METHOD PUBLIC finish : BOOL//Return value = TRUE if state was <> 0 and Err.flag = FALSE
VAR_INPUT
END_VAR
IF state <> 0 
THEN
	Busy 													:= FALSE;
	Done 													:= NOT Err.flag;
	     													  													
	text 													:= CONCAT('FINISH~State:',DINT_TO_STRING(state));
	text 													:= CONCAT(text,'(SetState:');
	text 													:= CONCAT(text,DINT_TO_STRING(MemSetState));
	text 													:= CONCAT(text,')/Busy=');
	text 													:= CONCAT(text,BOOL_TO_STRING(Busy));
	text 													:= CONCAT(text,'/Done=');
	text 													:= CONCAT(text,BOOL_TO_STRING(Done));
	
	state													:= 0;
	Finish 													:= Done;	
ELSE
	Finish 													:= FALSE;
END_IF
END_METHOD

METHOD PUBLIC incState : BOOL //Increment State by NoOfIncrements / Result always true 
VAR_INPUT
	NoOfIncrements								:	DINT;
END_VAR
State := State + NoOfIncrements;
incState := TRUE;
END_METHOD

METHOD PUBLIC reset : BOOL //return value = TRUE if execution finished 
VAR_INPUT
END_VAR
Done 														:= FALSE;
Busy 														:= FALSE;
text 														:= CONCAT('RESET~State:',DINT_TO_STRING(state));
text 														:= CONCAT(text,'(SetState:');
text 														:= CONCAT(text,DINT_TO_STRING(MemSetState));
text 														:= CONCAT(text,')/Busy=');
text 														:= CONCAT(text,BOOL_TO_STRING(Busy));
text 														:= CONCAT(text,'/Done=');
text 														:= CONCAT(text,BOOL_TO_STRING(Done));

MemSetState := state 										:=  0;
reset 														:= TRUE;
END_METHOD

METHOD PUBLIC resetWithErrHdl : BOOL //return value = TRUE if execution finished 
VAR_INPUT
END_VAR
Reset();
Err.Reset();
ResetWithErrHdl												 := TRUE;
END_METHOD

METHOD PUBLIC set : BOOL //Set MemSetstate to state value, Return value = TRUE if sequence handle will be busy (State <> 0)
VAR_INPUT
	State													:		 DINT;
END_VAR
MemSetState 												:= THIS^.state := State;
Busy 														:= state <> 0;
Done 														:= FALSE;
Set															:= Busy;
                    										
text 														:= CONCAT('SET~State:',DINT_TO_STRING(MemSetstate));
END_METHOD

PROPERTY PUBLIC ton_BT : TIME
GET
IF ton.IN
	AND NOT ton.Q
THEN
	Ton_BT 													:= ton.PT - ton.ET;
ELSE       													
	Ton_BT 													:= T#0MS;
END_IF
END_GET
END_PROPERTY

PROPERTY PUBLIC ton_PT : TIME
GET
Ton_PT 														:= ton.PT;
END_GET
SET
PUBLIC 
VAR
END_VAR
Ton.PT 														:= Ton_PT;
END_SET
END_PROPERTY

METHOD PUBLIC tonOFF : BOOL //Return value = TRUE if execution finished
VAR_INPUT
END_VAR
TON(In := FALSE,Q => );
TonOFF := NOT Ton.Q;
END_METHOD

METHOD PUBLIC tonON : BOOL; //Return value = TRUE if execution finished
VAR_INPUT
END_VAR
TON(In := TRUE,Q => TonON);
END_METHOD

METHOD PUBLIC tonRUN : BOOL //Return value status of time (Ton.Q)
VAR_INPUT
	IN														:	BOOL;
	PT														:	TIME;
END_VAR
THIS^.TON.IN := IN;
THIS^.TON.PT := PT;
TON(IN := IN , PT := PT, Q => TonRUN);
END_METHOD

END_FUNCTION_BLOCK

// POUs/_Miscellaneous/setNoOfBits
//Returns a LWORD variable with number (no) of bits set to TRUE starting from lowest significant bit (.0)  
{attribute 'displaymode':='binary'}		
FUNCTION setNoOfBits : LWORD 
VAR_INPUT
	No														:	INT;
END_VAR
VAR
	u64														:	U_64BIT_DATATYPE;
END_VAR

IF No <= 0
THEN
	setNoOfBits												:= 0;
ELSIF No <= 32
THEN
	setNoOfBits												:= TO_LWORD((EXPT(2,No) - 1));
ELSE
	u64._DWORDs[0]											:= 16#FFFFFFFF;
	u64._DWORDs[1]											:= TO_DWORD((EXPT(2,No - 32) - 1));
	setNoOfBits												:= u64._LWORD;
END_IF

END_FUNCTION

// POUs/_Miscellaneous/TEST_FB
//Should be called after new FBs to test signal flow and behavior of PlcOpen related variables 
FUNCTION_BLOCK Test_FB
VAR_OUTPUT CONSTANT
	NO_ERR 													:	INT := 0;
 	OK														:	INT := 1;
	ERR_BUSY 												:	INT := 2;
	ERR_DONE 												:	INT := 3;	
	ERR_ERR 												:	INT := 4;
	ERR_DONE_ERROR											:	INT := 5;
	ERR_NO_SIGNAL											:	INT := 6;
END_VAR             										
VAR_INPUT           										
	Reset													:	BOOL;	//The function block will be reset with a rising edge 
	Execute													:	BOOL;	//Link with Execute of the Fb to be tested
	Busy													:	BOOL;	//link with Busy Output of FB to be tested
	Error													:	BOOL;	//link with Error Output of FB to be tested
	Done													:	BOOL;	//link with Done Output of FB to be tested
END_VAR
VAR_OUTPUT
	ErrorId			:	INT := 0;	//Error identification 
END_VAR
VAR
	state			:	INT;
END_VAR

IF Reset
THEN
	state 													:= 0;
	ErrorId 												:= NO_ERR;
ELSE

	CASE state OF
	0:
		IF Execute
		THEN
			Errorid 										:= NO_ERR;
			IF Busy     									
			THEN        									
				state 										:= 10;
			ELSIF Error 									
			THEN        									
				state 										:= 20;
			ELSE        									
				state										:= state * -1;
				ErrorId 									:= ERR_BUSY;
			END_IF
		END_IF

	10:
		IF NOT Busy
		THEN
			IF Done
				AND Error
			THEN
				state										:= state * -1;
				ErrorId 									:= ERR_DONE_ERROR;
			ELSIF Done
			THEN
				IF Execute
				THEN
					state 									:= 11;
				ELSE      									
					state 									:= 12;
				END_IF
			ELSIF Error
			THEN
				IF Execute
				THEN
					state 									:= 21;
				ELSE      									
					state 									:= 22;
				END_IF
			ELSE
				state										:= state * -1;
				ErrorId 									:= ERR_NO_SIGNAL;
			END_IF
		END_IF

	11: (* Done muss wegsein wenn Execute nicht mehr da *)
		IF NOT Execute
		THEN
			IF NOT Done
			THEN
				state										:= 99;
			ELSE                							
				state										:= state * -1;
				ErrorId 									:= ERR_DONE;
			END_IF
		END_IF

	12: (* Done muss wegsein weil nur ein Zyklus *)
		IF NOT Done
		THEN
			state 											:= 99;
		ELSE
			state											:= state * -1;
			ErrorId 										:= ERR_DONE;
		END_IF


	20: (* Error Ohne Busy *)
		IF NOT Execute
		THEN
			IF Done
			THEN
				state										:= state * -1;
				ErrorId 									:= ERR_DONE;
			ELSIF Busy          							
			THEN                							
				state										:= state * -1;
				ErrorId 									:= ERR_BUSY;
			ELSE                	
				state										:= 99;
			END_IF
		END_IF

	21: (* Error muss wegsein wenn Execute nicht mehr da *)
		IF NOT Execute
		THEN
			IF NOT Error
			THEN
				state									:= 99;
			ELSE                						
				state									:= state * -1;
				ErrorId 								:= ERR_ERR;
			END_IF
		END_IF


	22: (* Error muss wegsein weil nur ein Zyklus *)
		IF NOT Error
		THEN
			state 										:= 99;
		ELSE                							
			state										:= state * -1;
			ErrorId 									:= ERR_DONE;
		END_IF              							
                            							
                            	
	99:                     	
		ErrorId											:= OK;
		state											:= 0;

	ELSE
		;
	END_CASE


END_IF

END_FUNCTION_BLOCK

// POUs/IO/Output
{attribute 'no_check'}
//Simple object for one hardware output with an additionl bit to forward the Out status to the AT  %Q* variable
FUNCTION_BLOCK Output 
VAR_INPUT
	Enable													:	BOOL := TRUE;	//FB will be processed as long as enable is TRUE 	
	Out														:	BOOL := FALSE;	//sets output
END_VAR         								
VAR_OUTPUT      								
	status													:	BYTE := 0;		//query Options (conditions see below)
	Q												AT  %Q* :	BOOL;			//hardware output
END_VAR         							
VAR             				
END_VAR

IF Out THEN
	switchOn();
ELSE
	SwitchOff();
END_IF

status.0 													:= NOT Q;
status.1 													:= Q;
status.5 													:= Enable;

METHOD PUBLIC switchOff : booL
VAR_INPUT
END_VAR
Q := Out											:= FALSE;
SwitchOff											:= TRUE;
END_METHOD

METHOD PUBLIC switchOn : booL
VAR_INPUT
END_VAR
Out														:= TRUE;
SwitchOn := Q 											:= Enable AND Out;
END_METHOD

END_FUNCTION_BLOCK

// POUs/_Miscellaneous/TOGGLE
{attribute 'no_check'}
//Toggle / FlipFlop
FUNCTION_BLOCK TOGGLE
VAR_INPUT
	IN														:	BOOL;
	RST														:	BOOL;
END_VAR             										
VAR_OUTPUT          										
	Q														:	BOOL;
END_VAR             	
VAR                 	
	M														:	BOOL;
END_VAR

	(* Toggle 				             	 																*)
	(************************************************************************************)

(* Ablauf ********************************************************************)
IF IN
	AND NOT M
THEN
	Q														:= NOT Q;
END_IF
M															:=	IN;
IF RST 
THEN 
	Reset(); 
END_IF


(********************************************************************************)

METHOD PUBLIC CLK : BOOL //Return value = status of output Q
VAR_INPUT
END_VAR
Q															:= NOT Q; 														
CLK 														:= Q;
END_METHOD

METHOD RESET : BOOL //Return value = TRUE if execution finished
VAR_INPUT
END_VAR
M := Q := FALSE;
RESET	:= TRUE;
END_METHOD

METHOD PUBLIC SET : BOOL  //Return value = TRUE if execution finished
VAR_INPUT
END_VAR
SET := M := Q := TRUE;
END_METHOD

END_FUNCTION_BLOCK

// POUs/BoundsCheck/boundsError
//Result is TRUE if INT index is out of range
{attribute 'no_check'}
FUNCTION boundsError : BOOL
VAR_INPUT
	Index													:INT;
	Lower													:INT;
	Upper													:INT;
END_VAR                 								
VAR
END_VAR

BoundsError:=index < lower OR index > upper;

END_FUNCTION

// POUs/BoundsCheck/boundsOK
//Result is TRUE if INT index is inside the range
{attribute 'no_check'}
FUNCTION boundsOK : BOOL
VAR_INPUT
	Index													: INT;
	Lower													: INT;
	Upper													: INT;
END_VAR

BoundsOK:= index >= lower AND index <= upper;

END_FUNCTION

// POUs/BoundsCheck/CheckBoundsInfo
//CheckBoundsInfo creates a an message entry in the TwinCAT logger 
//and provides information about the number of bounds errors as well signal variables if an error occured.
//Example of TwinCAT logger message: 	'Array index too low! Lower: 1 Upper: 10 Index: 11'
//
//please copy code example for CheckBounds as shown at this code section below into your "CheckBounds (FUN)"
{attribute 'no_check'}
FUNCTION_BLOCK CheckBoundsInfo
VAR_INPUT
	Interlock												:	BOOL; //TestAndSet interlock for multicore use
END_VAR                 									
VAR_OUTPUT              									
	LogMsg													:	T_MAXSTRING; 	//Last ADS log message
	CountUpper												:	UDINT := 0; 	//Counter of CheckBounds errors if index is greater the the upper limit 
	CountLower												:	UDINT := 0;		//Counter of CheckBounds errors if index is smaller the the lower limit 
	ErrorUpper												:	BOOL;			//Error upper limit occured - see LogMsg for further information
	ErrorLower												:	BOOL;			//Error lower limit occured - see LogMsg for further information
END_VAR                 									
VAR                     	
	MEM														:	ARRAY[1..3] OF DINT;
END_VAR

(* 
//Code template for implicit check function of "CheckBounds (FUN)"
IF  index < lower 
THEN
	(* Return right index *)
	CheckBounds 											:= lower;	

	IF TestAndSet(ET.CheckBoundsInfo.Interlock)
	THEN
		ET.CheckBoundsInfo.SetErrorLower(index,lower,upper);
		ET.CheckBoundsInfo.Interlock						:= FALSE;
	END_IF

ELSIF index > upper 
THEN
	(* Return right index *)
	CheckBounds 											:= upper;
	
	IF TestAndSet(ET.CheckBoundsInfo.Interlock)
	THEN
		ET.CheckBoundsInfo.SetErrorUpper(index,lower,upper);
		ET.CheckBoundsInfo.Interlock						:= FALSE;
	END_IF
	
ELSE  
	CheckBounds 											:= index;
END_IF
*)

METHOD PUBLIC reset : BOOL //Return value = TRUE if execution finished
VAR_INPUT
END_VAR
IF 	ErrorUpper OR ErrorLower
THEN
	CountUpper 												:= CountLower := 0;
	ErrorUpper												:= FALSE;
	ErrorLower												:= FALSE;
	MEMSET(ADR(MEM),0,SIZEOF(MEM));
END_IF
reset														:= TRUE;
END_METHOD

METHOD PUBLIC setErrorLower : booL //called by implicit function CheckBounds
VAR_INPUT
	index, lower, upper: DINT;
END_VAR
LogMsg														:=CONCAT('Array index too low! Index:',DINT_TO_STRING(index));
LogMsg														:=CONCAT(LogMsg,', Lower:');
LogMsg														:=CONCAT(LogMsg,DINT_TO_STRING(Lower));
LogMsg														:=CONCAT(LogMsg,', Upper:');
LogMsg														:=CONCAT(LogMsg,DINT_TO_STRING(Upper));
                                                        	
CountLower 													:= CountLower +1;                                                   	
ErrorLower													:= TRUE;
                                                        	
// write daten into eventlogger                         	
IF	lower <> MEM[1]                                     	
	OR Upper <> MEM[2]                                  	
	OR Index <> MEM[3]                                  	
THEN                                                    	
	ADSLOGDINT(	ADSLOG_MSGTYPE_ERROR OR ADSLOG_MSGTYPE_LOG,
				LogMsg,
				0);
END_IF

// store errors in memorybuffer
MEM[1] 														:= lower;
MEM[2] 														:= Upper;
MEM[3] 														:= index;

setErrorLower												:= TRUE;
END_METHOD

METHOD PUBLIC setErrorUpper :booL//called by implicit function CheckBounds
VAR_INPUT
	index, lower, upper: DINT;
END_VAR
LogMsg															:=CONCAT('Array index too high! Index:',DINT_TO_STRING(index));
LogMsg															:=CONCAT(LogMsg,', Lower:');
LogMsg															:=CONCAT(LogMsg,DINT_TO_STRING(Lower));
LogMsg															:=CONCAT(LogMsg,', Upper:');
LogMsg															:=CONCAT(LogMsg,DINT_TO_STRING(Upper));

CountUpper 														:= CountUpper +1;
ErrorUpper														:= TRUE;

// write daten into eventlogger
IF lower <> MEM[1]
	OR Upper <> MEM[2]
	OR Index <> MEM[3]
THEN
	ADSLOGDINT(	ADSLOG_MSGTYPE_ERROR OR ADSLOG_MSGTYPE_LOG,
					LogMsg,
					0);
END_IF

// store errors in memorybuffer
MEM[1] 															:= lower;
MEM[2] 															:= Upper;
MEM[3] 															:= index;

setErrorUpper													:= TRUE;
END_METHOD

END_FUNCTION_BLOCK

// POUs/Connectivity/ADS/AdsDataExchange
//"DataExchange" enables a ADS communication by symbol name between two TwinCAT runtime system
//based on Tc2_System
{attribute 'no_check'}
FUNCTION_BLOCK AdsDataExchange
VAR_OUTPUT CONSTANT
	MODE_FETCH_CONTINOUS									:	INT := 0;
	MODE_FETCH_BY_EVENT										:	INT := 1;
	MODE_SEND_CONTINOUS										:	INT := 2;
	MODE_SEND_BY_EVENT										:	INT := 3;
END_VAR
VAR_IN_OUT
END_VAR
VAR_INPUT
	Enable													:	BOOL := FALSE;	// FB will be processed as long as enable is TRUE 
	Transmit												:	BOOL := FALSE;	// TRUE or a rising edge starts the data exchange - depends on requested mode 
	Mode													:	INT (MODE_FETCH_CONTINOUS..MODE_SEND_BY_EVENT ) := MODE_SEND_BY_EVENT; //requested modes
	NetId													:	T_AmsNetId := ''; // Target AMS-NetID or '' for local-target
	Port													:	T_AmsPort := 851; 	// ADS-Communication-Port (PLC Runtime Port)
	DestSymbol												:	STRING;			//Desination symbol name to fetch or send - depends on requested mode
	pData													:	PVOID := 0;		//Pointer of data to send or target to fetch data - depends on requested mode 
	cbData													:	UDINT := 0;		//Data size of data to send or target to fetch data - depends on requested mode 
	Timeout													:	TIME := DEFAULT_ADS_TIMEOUT;// timeout for ADS request
END_VAR
VAR_OUTPUT
	hSymbol													:	UDINT;	//Symbol handle
	Ready													:	BOOL;	//ADS Route initialized successfully and ready to send/fetch											
	Active													:	BOOL;	//communication data exchange is in process (transmit triggered=
	Busy													:	BOOL; 	//Busy is TRUE at the rising edge of Enable and stays TRUE as long as the FB is performing any action. 
	Error													:	BOOL;	//Rising edge of Error informs that an error occurred during the execution of the Function Block  
{attribute 'displaymode':='hex'}
	ErrorID													:	UDINT; 	//Error identification - see ADS return codes at Beckhoff infosys for further information 
END_VAR
VAR
(* local variables *****************************************************)
	state													: 	INT := 0;
	MemErrorId												:	UDINT := 0;
	
(* trigger **********************************************************)
	FT_Enable												:	F_TRIG;
	RT_Transmit												:	R_TRIG;

(* timer ************************************************************)

(* finstances ***************************************************************)
	AdsRdWr_CreateVar_H										:	ADSRDWRT;
	FetchVal_ReqVar											:	ADSREAD;
	SendVal_ReqVar											:	ADSWRITE;
	ReleaseSymHandle										:	ADSWRITE;
END_VAR

FT_Enable(CLK 	:= Enable); // necessary for handle release 
RT_Transmit(CLK := Transmit AND Ready); // necessary for event mode

(* Sequence ********************************************************************************)
IF Enable THEN
	CASE state OF
	0: //Start creating symbol handle
		//Init fbs		
		AdsRdWr_CreateVar_H(WRTRD := FALSE);
		FetchVal_ReqVar(READ := FALSE);
		SendVal_ReqVar(WRITE := FALSE);
		ReleaseSymHandle(WRITE := FALSE);
		
		Busy 												:= TRUE;
		
		IF NOT AdsRdWr_CreateVar_H.BUSY AND NOT FetchVal_ReqVar.BUSY
			AND NOT SendVal_ReqVar.BUSY AND NOT ReleaseSymHandle.BUSY
		THEN
			AdsRdWr_CreateVar_H(NETID := NETID, PORT := PORT,
								IDXGRP := ADSIGRP_SYM_HNDBYNAME, IDXOFFS := 0,
								WRITELEN := SIZEOF(DestSymbol),// max. no. of chars req. variable
								READLEN := SIZEOF(hSymbol),
								SRCADDR := ADR(DestSymbol)	, DESTADDR := ADR(hSymbol), WRTRD := TRUE, TMOUT := Timeout);
			state											:= state + 1;						
		END_IF


	1://Wait for symbol handle 
		AdsRdWr_CreateVar_H(NETID := NETID, PORT := PORT,
							IDXGRP := ADSIGRP_SYM_HNDBYNAME, IDXOFFS := 0,
							WRITELEN := SIZEOF(DestSymbol),// max. no. of chars req. variable
							READLEN := SIZEOF(hSymbol),
							SRCADDR := ADR(DestSymbol)	, DESTADDR := ADR(hSymbol), WRTRD := TRUE, TMOUT := Timeout);	
		IF NOT AdsRdWr_CreateVar_H.BUSY
		THEN
			IF AdsRdWr_CreateVar_H.ERR
			THEN
				Busy										:= FALSE;
				Error										:= TRUE;
				ErrorId										:= AdsRdWr_CreateVar_H.ERRID;
				state										:= state * -1;
			ELSE
				Ready										:= TRUE;
				state										:= state + 1;
			END_IF
			AdsRdWr_CreateVar_H(WRTRD := FALSE);
		END_IF
		
	2: //Start fetch or send data 
		IF RT_Transmit.Q AND Mode = MODE_FETCH_BY_EVENT 
			OR Mode = MODE_FETCH_CONTINOUS
		THEN	
		 	FetchVal_ReqVar(	
				NETID 	:= NETID, 
				PORT 	:= PORT, 
				TMOUT 	:= Timeout,
				IDXGRP 	:= ADSIGRP_SYM_VALBYHND, 
				IDXOFFS := hSymbol, 	
				LEN 	:= cbData, 	
				DESTADDR:= pData,
				READ 	:= TRUE);
			Active											:= TRUE;
			state											:= state + 1;
		ELSIF RT_Transmit.Q AND Mode = MODE_SEND_BY_EVENT 
			OR Mode = MODE_SEND_CONTINOUS
		THEN 
			SendVal_ReqVar( 
				NETID 	:= NETID, 
				PORT 	:= PORT, 
				TMOUT 	:= Timeout,
				IDXGRP 	:= ADSIGRP_SYM_VALBYHND, 
				IDXOFFS	:= hSymbol, 
				SRCADDR := pData,
				LEN		:= cbData,  
				WRITE 	:= TRUE);		
			Active											:= TRUE;
			state											:= state + 1;
		END_IF
		
	3: //Wait for send/fetch done 
		IF FetchVal_ReqVar.READ
		THEN
		 	FetchVal_ReqVar(LEN 	:= cbData, DESTADDR:= pData, READ 	:= TRUE);		
			IF NOT FetchVal_ReqVar.BUSY
			THEN
				Active										:= FALSE;
				IF FetchVal_ReqVar.ERR
				THEN
					Busy									:= FALSE;
					Error									:= TRUE;
					ErrorId									:= FetchVal_ReqVar.ERRID;
					state									:= state * -1;					
				ELSE
					Ready									:= TRUE;
					state 									:= state - 1;
				END_IF
				FetchVal_ReqVar(READ 	:= FALSE);
			END_IF
		
		ELSE
			SendVal_ReqVar( SRCADDR := pData,LEN := cbData,  WRITE 	:= TRUE);	
			IF NOT SendVal_ReqVar.BUSY
			THEN		
				Active										:= FALSE;
				IF SendVal_ReqVar.ERR
				THEN
					Busy									:= FALSE;
					Error									:= TRUE;
					ErrorId									:= SendVal_ReqVar.ERRID;
					state									:= state * -1;					
				ELSE
					Ready									:= TRUE;
					state 									:= state - 1;
				END_IF
				SendVal_ReqVar(WRITE 	:= FALSE);		
			END_IF
		END_IF
	ELSE //Error - wait for enable = FALSE	
		MemErrorId											:= ErrorId;
 	END_CASE
ELSE //Enable = FALSE	
	Active													:= FALSE;
	Ready													:= FALSE;
	IF FT_Enable.Q 
	THEN  
		ReleaseSymHandle(WRITE:= FALSE);
		ReleaseSymHandle(NETID := NETID, 
						PORT 	:= PORT, 
						TMOUT 	:= Timeout,
						IDXGRP 	:= ADSIGRP_SYM_RELEASEHND, 
						IDXOFFS := hSymbol, 
						LEN 	:= 0, 
						WRITE 	:= hSymbol <> 0);
	ELSE
		ReleaseSymHandle();
		IF NOT ReleaseSymHandle.BUSY
		THEN
			ReleaseSymHandle(Write := FALSE);
			hSymbol											:= 0;
			Error 											:= FALSE;		
			ErrorID 										:= 0;
			Busy 											:= FALSE;
			State	 										:= 0;				
		END_IF
	END_IF

END_IF
	
(*********************************************************************************************************)

END_FUNCTION_BLOCK

// POUs/Connectivity/TF625x-Modbus/Master/_Components/ModbusJob
{attribute 'no_check'}
// description of Slave Job (data structure)
FUNCTION_BLOCK ModbusJob	
VAR_INPUT
	FunctionCode		:	BYTE;
	StartAddress		:	WORD;
	Quantity			:	WORD;
	Valid				:	BOOL;
	Timestamp			:	DATE_AND_TIME;
END_VAR
VAR_OUTPUT
END_VAR
VAR
END_VAR

;

METHOD PUBLIC init : BOOL //Return value = TRUE if execution finished
VAR_INPUT
END_VAR
	functionCode											:= 0;
	startAddress											:= 0;
	valid													:= FALSE;
	MEMSET(ADR(quantity), 16#0, SIZEOF(quantity));	
	MEMSET(ADR(timeStamp), 16#0, SIZEOF(timeStamp));
	Init													:= TRUE;
END_METHOD

END_FUNCTION_BLOCK

// POUs/Connectivity/TF625x-Modbus/Master/_Components/ModbusSlaveCom
{attribute 'no_check'}
//communication struct between modbus master FB and Slave FB
FUNCTION_BLOCK ModbusSlaveCom 
VAR_OUTPUT CONSTANT
	MIN_SLAVE_JOB			:	INT := 1;
	MAX_SLAVE_JOB			:	INT := PARAM.MODBUS_MAX_SLAVE_JOB;
	MIN_DATA				:	INT := 1;
	MAX_DATA				:	INT := 120;
END_VAR                 	
VAR_INPUT               	
	Enable					:	BOOL;
	writeJobRequested		:	BOOL;
	IpAddr 					:	T_IPv4Addr;	// use only for TCP and UDP or ''		// use only for TCP and UDP 
	Port 					:	UDINT;			// use only for TCP
	Address					:	BYTE;
	NoOfJobs				:	INT;
	Jobs					:	ARRAY[MIN_SLAVE_JOB..MAX_SLAVE_JOB] OF ModbusJob;
	Data					:	ARRAY[MIN_DATA..MAX_DATA] OF WORD;
	CurrentJobIdx			:	INT 	:= 1;
	CountGood				:	DWORD 	:= 0;
	CountBad				:	DWORD 	:= 0;
END_VAR
VAR_OUTPUT
END_VAR
VAR
END_VAR

;

METHOD PUBLIC deleteData : booL //Return value = TRUE if execution finished
VAR_INPUT
END_VAR
MEMSET(ADR(Data),0,SIZEOF(Data));
DeleteData := TRUE;
END_METHOD

END_FUNCTION_BLOCK

// POUs/Connectivity/TF625x-Modbus/Master/TF6250-ModbusTcpServer/TCP/ModbusTcpMaster
{attribute 'no_check'}
// ModBus comunication master to multible slaves useing TCP protocol	
// based on TF6250 - required lib: Tc2_ModbusTCP
FUNCTION_BLOCK ModbusTcpMaster
VAR CONSTANT
	MIN_SLAVE												:	INT := 1;
	MAX_SLAVE												:	INT := PARAM.MODBUS_MAX_SLAVES_OF_MASTER;
END_VAR
VAR_INPUT
	Enable													:	BOOL ; 	// FB will be processed as long as enable is TRUE 
	ResetTrig												:	BOOL ; 	// The function block will be reset with a rising edge 
	SlaveCom												:	ARRAY[MIN_SLAVE..MAX_SLAVE] OF POINTER TO ModbusSlaveCom;
	Timestamp												:	DT;
END_VAR         	
VAR_OUTPUT      	
	JobNo													:	INT := 0;
	SlaveNo													:	INT := 0;
	Error													:	BOOL; 	// Rising edge of Error informs that an error occurred during the execution of the Function Block 
{attribute 'displaymode':='hex'}
	ErrorID													:	UDINT; 	// Error identification - see ADS return codes at Beckhoff infosys for further information 
	ErrorText												:	STRING;
END_VAR
VAR
(* memory **************************************************)
	state 													:	INT := 0;

(* trigger *************************************************)

(* timer ***************************************************)

(* blocks **************************************************)
	ReadCoils												:	FB_MBReadCoils := (tTimeout	 := DEFAULT_ADS_TIMEOUT);			// Fnc 1
	ReadInputs												:	FB_MBReadInputs := (tTimeout := DEFAULT_ADS_TIMEOUT);			// Fnc 2
	ReadRegs												:	FB_MBReadRegs := (tTimeout	:= DEFAULT_ADS_TIMEOUT);			// Fnc 3
	ReadInputRegs											:	FB_MBReadInputRegs := (tTimeout	:= DEFAULT_ADS_TIMEOUT);		// Fnc 4
	WriteSingleCoil											:	FB_MBWriteSingleCoil := (tTimeout	:= DEFAULT_ADS_TIMEOUT);	// Fnc 5
	WriteSingleReg											:	FB_MBWriteSingleReg := (tTimeout:= DEFAULT_ADS_TIMEOUT);		// Fnc 6
	Diagnose												:	FB_MBDiagnose := (tTimeout	:= DEFAULT_ADS_TIMEOUT);			// Fnc 8
	WriteCoils												:	FB_MBWriteCoils := (tTimeout:= DEFAULT_ADS_TIMEOUT);			// Fnc 15
	WriteRegs												:	FB_MBWriteRegs := (tTimeout	:= DEFAULT_ADS_TIMEOUT);			// Fnc 16
	ReadWriteRegs											:	FB_MBReadWriteRegs := (tTimeout	:= DEFAULT_ADS_TIMEOUT); 		// Fnc 23	use read and write job instead
(* internal used variables *********************************)
	i,j,k													:	INT :=0;
END_VAR


	CASE state OF
	0:	(* Idle *)
		IF Enable 
		THEN
			k 												:=	0;
			JobNo  :=  SlaveNo								:=	1;
			state 											:=	10;
		END_IF

	10: 
		IF GetNextSlave() 
		THEN (* find Slave *)
			k 												:= 0;
			IF GetNextJob() 
			THEN (* find JobNo *)
				SlaveCom[SlaveNo]^.currentJobIdx 			:= JobNo;
				SlaveCom[SlaveNo]^.writeJobRequested 		:= SlaveCom[SlaveNo]^.Jobs[JobNo].FunctionCode >= 5;
				State 										:= SEL(SlaveCom[SlaveNo]^.writeJobRequested, 20, 15);
			END_IF
		ELSE
			state 											:=	0;
		END_IF
			
	15: (* wait for valid write date *)
		IF NOT SlaveCom[SlaveNo]^.writeJobRequested
		THEN
			SlaveCom[SlaveNo]^.Jobs[JobNo].Valid 			:= FALSE;
			state 											:= 20;
		END_IF

	20: (* start job *)	
		IF NOT StartJob(FALSE) // Busy
		THEN						
			state 											:= 30;
		END_IF

	30: (* wait for com cycle *)
		IF NOT StartJob(TRUE) THEN // Busy
			IF Error 
			THEN
				ErrorText									:= CONCAT('Error at SlaveNo: ',	CONCAT(INT_TO_STRING(SlaveNo), CONCAT(', JobNo: ', INT_TO_STRING(JobNo))));
				SlaveCom[SlaveNo]^.countBad 				:= SlaveCom[SlaveNo]^.countBad +1;
				state 										:= 98; 
			ELSE
				SlaveCom[SlaveNo]^.countGood 				:= SlaveCom[SlaveNo]^.countGood +1;
				SlaveCom[SlaveNo]^.Jobs[JobNo].Valid 		:= TRUE;
				SlaveCom[SlaveNo]^.Jobs[JobNo].TimeStamp 	:= Timestamp;
				JobNo 										:= JobNo + 1;
				state 										:= 10;	(* next job *)
			END_IF
			StartJob(FALSE);
		END_IF

	98: (* wait for quit *)
		IF ResetTrig THEN
			reset();
		END_IF

	END_CASE

METHOD PRIVATE getNextJob : Bool //Return value = TRUE if execution finished
VAR_INPUT
END_VAR
	
	WHILE SlaveCom[SlaveNo]^.Jobs[JobNo].FunctionCode = 0 DO
		JobNo 											:= JobNo + 1;
		IF JobNo > SlaveCom[SlaveNo]^.MAX_SLAVE_JOB THEN
			JobNo 										:= SlaveCom[SlaveNo]^.MIN_SLAVE_JOB;
			SlaveNo 									:= SlaveNo + 1;
			GetNextJob									:= FALSE;
			RETURN;
		END_IF
	END_WHILE
	GetNextJob											:= TRUE;
END_METHOD

METHOD PRIVATE getNextSlave : Bool //Return value = TRUE if execution finished
VAR_INPUT
END_VAR
	WHILE SlaveCom[SlaveNo] = 0 OR_ELSE NOT SlaveCom[SlaveNo]^.Enable DO
		SlaveNo 										:= SlaveNo + 1;
		IF SlaveNo > MAX_SLAVE 
		THEN
			k 											:= k + 1;
			SlaveNo 									:= MIN_SLAVE;
		ELSIF k = 2 
		THEN
			k 											:= 0;
			GetNextSlave								:= FALSE;
			RETURN;
		END_IF	
	END_WHILE
	GetNextSlave										:= TRUE;
END_METHOD

METHOD PUBLIC reset : bool //Return value = TRUE if execution finished
VAR_INPUT
END_VAR
IF State = 98 
THEN
	Error													:= FALSE;
	ErrorID													:= 0;
	ErrorText												:= '';
	state													:= 0;
END_IF
reset														:= TRUE;
END_METHOD

METHOD PRIVATE startJob : BOOL //Return value = TRUE as long as the job is busy
VAR_INPUT
	Execute							: BOOL;
END_VAR
	IF 		SlaveCom[SlaveNo]^.Jobs[JobNo].FunctionCode = 1 THEN
		ReadCoils(
			sIPAddr			:= SlaveCom[SlaveNo]^.ipAddr, 
			nTCPPort		:= TO_UINT(SlaveCom[SlaveNo]^.Port), 
			nUnitID			:= SlaveCom[SlaveNo]^.Address, 
			nQuantity		:= SlaveCom[SlaveNo]^.jobs[JobNo].Quantity, 
			nMBAddr			:= SlaveCom[SlaveNo]^.jobs[JobNo].startAddress, 
			cbLength		:= SlaveCom[SlaveNo]^.jobs[JobNo].Quantity, 
			pDestAddr		:= ADR(SlaveCom[SlaveNo]^.Data), 
			bExecute		:= Execute, 
			tTimeout		:= , 
			bBusy			=> StartJob, 
			bError			=> Error, 
			nErrId			=> ErrorID);
			
	ELSIF 	SlaveCom[SlaveNo]^.Jobs[JobNo].FunctionCode = 2 THEN
		ReadInputs(
			sIPAddr			:= SlaveCom[SlaveNo]^.ipAddr, 
			nTCPPort		:= TO_UINT(SlaveCom[SlaveNo]^.Port), 
			nUnitID			:= SlaveCom[SlaveNo]^.Address, 
			nQuantity		:= SlaveCom[SlaveNo]^.jobs[JobNo].Quantity, 
			nMBAddr			:= SlaveCom[SlaveNo]^.jobs[JobNo].startAddress, 
			cbLength		:= SlaveCom[SlaveNo]^.jobs[JobNo].Quantity, 
			pDestAddr		:= ADR(SlaveCom[SlaveNo]^.Data), 
			bExecute		:= Execute, 
			tTimeout		:= , 
			bBusy			=> StartJob, 
			bError			=> Error, 
			nErrId			=> ErrorID);
			
	ELSIF 	SlaveCom[SlaveNo]^.Jobs[JobNo].FunctionCode = 3 THEN
		ReadRegs(
			sIPAddr			:= SlaveCom[SlaveNo]^.ipAddr, 
			nTCPPort		:= TO_UINT(SlaveCom[SlaveNo]^.Port), 
			nUnitID			:= SlaveCom[SlaveNo]^.Address, 
			nQuantity		:= SlaveCom[SlaveNo]^.jobs[JobNo].Quantity, 
			nMBAddr			:= SlaveCom[SlaveNo]^.jobs[JobNo].startAddress, 
			cbLength		:= SlaveCom[SlaveNo]^.jobs[JobNo].Quantity * 2, 
			pDestAddr		:= ADR(SlaveCom[SlaveNo]^.Data), 
			bExecute		:= Execute, 
			tTimeout		:= , 
			bBusy			=> StartJob, 
			bError			=> Error, 
			nErrId			=> ErrorID);
	
	ELSIF 	SlaveCom[SlaveNo]^.Jobs[JobNo].FunctionCode = 4 THEN
		ReadInputRegs(
			sIPAddr			:= SlaveCom[SlaveNo]^.ipAddr, 
			nTCPPort		:= TO_UINT(SlaveCom[SlaveNo]^.Port), 
			nUnitID			:= SlaveCom[SlaveNo]^.Address, 
			nQuantity		:= SlaveCom[SlaveNo]^.jobs[JobNo].Quantity, 
			nMBAddr			:= SlaveCom[SlaveNo]^.jobs[JobNo].startAddress, 
			cbLength		:= SlaveCom[SlaveNo]^.jobs[JobNo].Quantity * 2, 
			pDestAddr		:= ADR(SlaveCom[SlaveNo]^.Data), 
			bExecute		:= Execute, 
			tTimeout		:= , 
			bBusy			=> StartJob, 
			bError			=> Error, 
			nErrId			=> ErrorID);
	
	ELSIF 	SlaveCom[SlaveNo]^.Jobs[JobNo].FunctionCode = 5 THEN
		WriteSingleCoil(
			sIPAddr			:= SlaveCom[SlaveNo]^.ipAddr, 
			nTCPPort		:= TO_UINT(SlaveCom[SlaveNo]^.Port), 
			nUnitID			:= SlaveCom[SlaveNo]^.Address, 
			nMBAddr			:= SlaveCom[SlaveNo]^.jobs[JobNo].startAddress, 
			nValue			:= SlaveCom[SlaveNo]^.data[1], 
			bExecute		:= Execute, 
			tTimeout		:= , 
			bBusy			=> StartJob, 
			bError			=> Error, 
			nErrId			=> ErrorID);
	
	ELSIF 	SlaveCom[SlaveNo]^.Jobs[JobNo].FunctionCode = 6 THEN
		WriteSingleReg(
			sIPAddr			:= SlaveCom[SlaveNo]^.ipAddr, 
			nTCPPort		:= TO_UINT(SlaveCom[SlaveNo]^.Port), 
			nUnitID			:= SlaveCom[SlaveNo]^.Address, 
			nMBAddr			:= SlaveCom[SlaveNo]^.jobs[JobNo].startAddress, 
			nValue			:= SlaveCom[SlaveNo]^.data[1], 
			bExecute		:= Execute, 
			tTimeout		:= , 
			bBusy			=> StartJob, 
			bError			=> Error, 
			nErrId			=> ErrorID);	
			
	ELSIF 	SlaveCom[SlaveNo]^.Jobs[JobNo].FunctionCode = 8 THEN
		Diagnose(
			sIPAddr			:= SlaveCom[SlaveNo]^.ipAddr, 
			nTCPPort		:= TO_UINT(SlaveCom[SlaveNo]^.Port), 
			nUnitID			:= SlaveCom[SlaveNo]^.Address, 
			bExecute		:= Execute, 
			tTimeout		:= , 
			bBusy			=> StartJob, 
			bError			=> Error, 
			nErrId			=> ErrorID);		

	ELSIF 	SlaveCom[SlaveNo]^.Jobs[JobNo].FunctionCode = 15 THEN
		WriteCoils(
			sIPAddr			:= SlaveCom[SlaveNo]^.ipAddr, 
			nTCPPort		:= TO_UINT(SlaveCom[SlaveNo]^.Port), 
			nUnitID			:= SlaveCom[SlaveNo]^.Address, 
			nQuantity		:= SlaveCom[SlaveNo]^.jobs[JobNo].Quantity, 
			nMBAddr			:= SlaveCom[SlaveNo]^.jobs[JobNo].startAddress, 
			cbLength		:= SlaveCom[SlaveNo]^.jobs[JobNo].Quantity, 
			pSrcAddr		:= ADR(SlaveCom[SlaveNo]^.Data), 
			bExecute		:= Execute, 
			tTimeout		:= , 
			bBusy			=> StartJob, 
			bError			=> Error, 
			nErrId			=> ErrorID);
	
	ELSIF 	SlaveCom[SlaveNo]^.Jobs[JobNo].FunctionCode = 16 THEN
		WriteRegs(
			sIPAddr			:= SlaveCom[SlaveNo]^.ipAddr, 
			nTCPPort		:= TO_UINT(SlaveCom[SlaveNo]^.Port), 
			nUnitID			:= SlaveCom[SlaveNo]^.Address, 
			nQuantity		:= SlaveCom[SlaveNo]^.jobs[JobNo].Quantity, 
			nMBAddr			:= SlaveCom[SlaveNo]^.jobs[JobNo].startAddress, 
			cbLength		:= SlaveCom[SlaveNo]^.jobs[JobNo].Quantity, 
			pSrcAddr		:= ADR(SlaveCom[SlaveNo]^.Data), 
			bExecute		:= Execute, 
			tTimeout		:= , 
			bBusy			=> StartJob, 
			bError			=> Error, 
			nErrId			=> ErrorID);
		
	ELSIF 	SlaveCom[SlaveNo]^.Jobs[JobNo].FunctionCode = 23 THEN
		// not implemented
(*		ReadWriteRegs(
			sIPAddr			:= SlaveCom[SlaveNo]^.ipAddr, 
			nTCPPort		:= SlaveCom[SlaveNo]^.Port, 
			nUnitID			:= SlaveCom[SlaveNo]^.Address, 
			nReadQuantity	:= SlaveCom[SlaveNo]^.jobs[JobNo].Quantity, 
			nMBReadAddr		:= SlaveCom[SlaveNo]^.jobs[JobNo].startAddress, 
			nWriteQuantity	:= , // missing
			nMBWriteAddr	:= , // missing
			cbDestLength	:= SlaveCom[SlaveNo]^.jobs[JobNo].Quantity, 
			pDestAddr		:= ADR(SlaveCom[SlaveNo]^.Data),
			cbSrcLength		:= , // missing
			pSrcAddr 		:= , // missing
			bExecute		:= Execute, 
			tTimeout		:= , 
			bBusy			=> StartJob, 
			bError			=> Error, 
			nErrId			=> ErrorID);	
		*)			
	END_IF
END_METHOD

END_FUNCTION_BLOCK

// POUs/Connectivity/TF625x-Modbus/Master/TF6250-ModbusTcpServer/UDP/ModbusUdpMaster
{attribute 'no_check'}
// ModBus comunication master to multible slaves useing UDP protocol
// based on TF6250 - required lib: Tc2_ModbusTCP
FUNCTION_BLOCK ModbusUdpMaster
VAR CONSTANT
	MIN_SLAVE												:	INT := 1;
	MAX_SLAVE												:	INT := PARAM.MODBUS_MAX_SLAVES_OF_MASTER;
END_VAR
VAR_INPUT
	Enable													:	BOOL ; 		// FB will be processed as long as enable is TRUE 
	ResetTrig												:	BOOL ;		// The function block will be reset with a rising edge 
	SlaveCom												:	ARRAY[MIN_SLAVE..MAX_SLAVE] OF POINTER TO ModbusSlaveCom;
	Timestamp												:	DT;
END_VAR         	
VAR_OUTPUT      	
	Error													:	BOOL;		// Rising edge of Error informs that an error occurred during the execution of the Function Block 
{attribute 'displaymode':='hex'}
	ErrorID													:	UDINT;		// Error identification - see ADS return codes at Beckhoff infosys for further information 
	ErrorText												:	STRING;
END_VAR
VAR
(* memory **************************************************)
	state 													:	INT := 0;
	JobNo													:	INT := 0;
	SlaveNo													:	INT := 0;
(* trigger *************************************************)

(* timer ***************************************************)

(* blocks **************************************************)
	ReadCoils												:	FB_MBUdpReadCoils := (tTimeout		:= DEFAULT_ADS_TIMEOUT);		// Fnc 1
	ReadInputs												:	FB_MBUdpReadInputs := (tTimeout		:= DEFAULT_ADS_TIMEOUT);		// Fnc 2
	ReadRegs												:	FB_MBUdpReadRegs := (tTimeout		:= DEFAULT_ADS_TIMEOUT);		// Fnc 3
	ReadInputRegs											:	FB_MBUdpReadInputRegs := (tTimeout	:= DEFAULT_ADS_TIMEOUT);	// Fnc 4
	WriteSingleCoil											:	FB_MBUdpWriteSingleCoil := (tTimeout:= DEFAULT_ADS_TIMEOUT);// Fnc 5
	WriteSingleReg											:	FB_MBUdpWriteSingleReg := (tTimeout	:= DEFAULT_ADS_TIMEOUT);	// Fnc 6
	Diagnose												:	FB_MBUdpDiagnose := (tTimeout		:= DEFAULT_ADS_TIMEOUT);		// Fnc 8
	WriteCoils												:	FB_MBUdpWriteCoils := (tTimeout		:= DEFAULT_ADS_TIMEOUT);		// Fnc 15
	WriteRegs												:	FB_MBUdpWriteRegs := (tTimeout		:= DEFAULT_ADS_TIMEOUT);		// Fnc 16
	ReadWriteRegs											:	FB_MBUdpReadWriteRegs := (tTimeout	:= DEFAULT_ADS_TIMEOUT); 	// Fnc 23	use read and write job instead
(* internal used variables *********************************)
	i,j,k													:	INT :=0;
END_VAR


	CASE state OF
	0:	(* Idle *)
		IF Enable 
		THEN
			k 												:=	0;
			JobNo  :=  SlaveNo								:=	1;
			state 											:=	10;
		END_IF

	10: 
		IF GetNextSlave() 
		THEN (* find Slave *)
			k 												:= 0;
			IF GetNextJob() 
			THEN (* find JobNo *)
				SlaveCom[SlaveNo]^.currentJobIdx 			:= JobNo;
				SlaveCom[SlaveNo]^.writeJobRequested 		:= SlaveCom[SlaveNo]^.Jobs[JobNo].FunctionCode >= 5;
				State 										:= SEL(SlaveCom[SlaveNo]^.writeJobRequested, 20, 15);
			END_IF
		ELSE
			state 											:=	0;
		END_IF
	
	15: (* wait for valid write date *)
		IF NOT SlaveCom[SlaveNo]^.writeJobRequested
		THEN
			SlaveCom[SlaveNo]^.Jobs[JobNo].Valid 			:= FALSE;
			state 											:= 20;
		END_IF

	20: (* start job *)	
		IF NOT StartJob(FALSE) // Busy
		THEN						
			state 											:= 30;
		END_IF

	30: (* wait for com cycle *)
		IF NOT StartJob(TRUE) THEN // Busy
			IF Error 
			THEN
				ErrorText									:= CONCAT('Error at SlaveNo: ',	CONCAT(INT_TO_STRING(SlaveNo), CONCAT(', JobNo: ', INT_TO_STRING(JobNo))));
				SlaveCom[SlaveNo]^.countBad 				:= SlaveCom[SlaveNo]^.countBad +1;
				state 										:= 98; 
			ELSE
				SlaveCom[SlaveNo]^.countGood 				:= SlaveCom[SlaveNo]^.countGood +1;
				SlaveCom[SlaveNo]^.Jobs[JobNo].Valid 		:= TRUE;
				SlaveCom[SlaveNo]^.Jobs[JobNo].TimeStamp 	:= Timestamp;
				JobNo 										:= JobNo + 1;
				state 										:= 10;	(* next job *)
			END_IF
			StartJob(FALSE);
		END_IF

	98: (* wait for quit *)
		IF ResetTrig THEN
			reset();
		END_IF

	END_CASE

METHOD PRIVATE getNextJob : Bool //Return value = TRUE if execution finished
VAR_INPUT
END_VAR
	
	WHILE SlaveCom[SlaveNo]^.Jobs[JobNo].FunctionCode = 0 DO
		JobNo 											:= JobNo + 1;
		IF JobNo > SlaveCom[SlaveNo]^.MAX_SLAVE_JOB THEN
			JobNo 										:= SlaveCom[SlaveNo]^.MIN_SLAVE_JOB;
			SlaveNo 									:= SlaveNo + 1;
			GetNextJob									:= FALSE;
			RETURN;
		END_IF
	END_WHILE
	GetNextJob											:= TRUE;
END_METHOD

METHOD PRIVATE getNextSlave : Bool //Return value = TRUE if execution finished
VAR_INPUT
END_VAR
	WHILE SlaveCom[SlaveNo] = 0 or_else not SlaveCom[SlaveNo]^.Enable DO
		SlaveNo 										:= SlaveNo + 1;
		IF SlaveNo > MAX_SLAVE 
		THEN
			k 											:= k + 1;
			SlaveNo 									:= MIN_SLAVE;
		ELSIF k = 2 
		THEN
			k 											:= 0;
			GetNextSlave								:= FALSE;
			RETURN;
		END_IF	
	END_WHILE
	GetNextSlave										:= TRUE;
END_METHOD

METHOD PUBLIC reset : booL //Return value = TRUE if execution finished
VAR_INPUT
END_VAR
IF State = 98 
THEN
	Error													:= FALSE;
	ErrorID													:= 0;
	ErrorText												:= '';
	state													:= 0;
END_IF	
reset														:= TRUE;
END_METHOD

METHOD PRIVATE startJob : BOOL //Return value = TRUE if busy - TRUE as long as the job is busy
VAR_INPUT
	Execute							: BOOL;
END_VAR
	IF 	SlaveCom[SlaveNo]^.Jobs[JobNo].FunctionCode = 1 THEN
		ReadCoils(
			sIPAddr			:= SlaveCom[SlaveNo]^.ipAddr, 
			nTCPPort		:= TO_UINT(SlaveCom[SlaveNo]^.Port), 
			nUnitID			:= SlaveCom[SlaveNo]^.Address, 
			nQuantity		:= SlaveCom[SlaveNo]^.jobs[JobNo].Quantity, 
			nMBAddr			:= SlaveCom[SlaveNo]^.jobs[JobNo].startAddress, 
			cbLength		:= SlaveCom[SlaveNo]^.jobs[JobNo].Quantity, 
			pDestAddr		:= ADR(SlaveCom[SlaveNo]^.Data), 
			bExecute		:= Execute, 
			tTimeout		:= , 
			bBusy			=> StartJob, 
			bError			=> Error, 
			nErrId			=> ErrorID);
		
	ELSIF 	SlaveCom[SlaveNo]^.Jobs[JobNo].FunctionCode = 2 THEN
		ReadInputs(
			sIPAddr			:= SlaveCom[SlaveNo]^.ipAddr, 
			nTCPPort		:= TO_UINT(SlaveCom[SlaveNo]^.Port), 
			nUnitID			:= SlaveCom[SlaveNo]^.Address, 
			nQuantity		:= SlaveCom[SlaveNo]^.jobs[JobNo].Quantity, 
			nMBAddr			:= SlaveCom[SlaveNo]^.jobs[JobNo].startAddress, 
			cbLength		:= SlaveCom[SlaveNo]^.jobs[JobNo].Quantity, 
			pDestAddr		:= ADR(SlaveCom[SlaveNo]^.Data), 
			bExecute		:= Execute, 
			tTimeout		:= , 
			bBusy			=> StartJob, 
			bError			=> Error, 
			nErrId			=> ErrorID);
			
	ELSIF 	SlaveCom[SlaveNo]^.Jobs[JobNo].FunctionCode = 3 THEN
		ReadRegs(
			sIPAddr			:= SlaveCom[SlaveNo]^.ipAddr, 
			nTCPPort		:= TO_UINT(SlaveCom[SlaveNo]^.Port), 
			nUnitID			:= SlaveCom[SlaveNo]^.Address, 
			nQuantity		:= SlaveCom[SlaveNo]^.jobs[JobNo].Quantity, 
			nMBAddr			:= SlaveCom[SlaveNo]^.jobs[JobNo].startAddress, 
			cbLength		:= SlaveCom[SlaveNo]^.jobs[JobNo].Quantity * 2, 
			pDestAddr		:= ADR(SlaveCom[SlaveNo]^.Data), 
			bExecute		:= Execute, 
			tTimeout		:= DEFAULT_ADS_TIMEOUT, 
			bBusy			=> StartJob, 
			bError			=> Error, 
			nErrId			=> ErrorID);
	
	ELSIF 	SlaveCom[SlaveNo]^.Jobs[JobNo].FunctionCode = 4 THEN
		ReadInputRegs(
			sIPAddr			:= SlaveCom[SlaveNo]^.ipAddr, 
			nTCPPort		:= TO_UINT(SlaveCom[SlaveNo]^.Port), 
			nUnitID			:= SlaveCom[SlaveNo]^.Address, 
			nQuantity		:= SlaveCom[SlaveNo]^.jobs[JobNo].Quantity, 
			nMBAddr			:= SlaveCom[SlaveNo]^.jobs[JobNo].startAddress, 
			cbLength		:= SlaveCom[SlaveNo]^.jobs[JobNo].Quantity * 2, 
			pDestAddr		:= ADR(SlaveCom[SlaveNo]^.Data), 
			bExecute		:= Execute, 
			tTimeout		:= , 
			bBusy			=> StartJob, 
			bError			=> Error, 
			nErrId			=> ErrorID);
	
	ELSIF 	SlaveCom[SlaveNo]^.Jobs[JobNo].FunctionCode = 5 THEN
		WriteSingleCoil(
			sIPAddr			:= SlaveCom[SlaveNo]^.ipAddr, 
			nTCPPort		:= TO_UINT(SlaveCom[SlaveNo]^.Port), 
			nUnitID			:= SlaveCom[SlaveNo]^.Address, 
			nMBAddr			:= SlaveCom[SlaveNo]^.jobs[JobNo].startAddress, 
			nValue			:= SlaveCom[SlaveNo]^.data[1], 
			bExecute		:= Execute, 
			tTimeout		:= , 
			bBusy			=> StartJob, 
			bError			=> Error, 
			nErrId			=> ErrorID);
	
	ELSIF 	SlaveCom[SlaveNo]^.Jobs[JobNo].FunctionCode = 6 THEN
		WriteSingleReg(
			sIPAddr			:= SlaveCom[SlaveNo]^.ipAddr, 
			nTCPPort		:= TO_UINT(SlaveCom[SlaveNo]^.Port), 
			nUnitID			:= SlaveCom[SlaveNo]^.Address, 
			nMBAddr			:= SlaveCom[SlaveNo]^.jobs[JobNo].startAddress, 
			nValue			:= SlaveCom[SlaveNo]^.data[1], 
			bExecute		:= Execute, 
			tTimeout		:= , 
			bBusy			=> StartJob, 
			bError			=> Error, 
			nErrId			=> ErrorID);
			
	ELSIF 	SlaveCom[SlaveNo]^.Jobs[JobNo].FunctionCode = 8 THEN
		Diagnose(
			sIPAddr			:= SlaveCom[SlaveNo]^.ipAddr, 
			nTCPPort		:= TO_UINT(SlaveCom[SlaveNo]^.Port), 
			nUnitID			:= SlaveCom[SlaveNo]^.Address, 
			bExecute		:= Execute, 
			tTimeout		:= , 
			bBusy			=> StartJob, 
			bError			=> Error, 
			nErrId			=> ErrorID);	
			
	ELSIF 	SlaveCom[SlaveNo]^.Jobs[JobNo].FunctionCode = 15 THEN
		WriteCoils(
			sIPAddr			:= SlaveCom[SlaveNo]^.ipAddr, 
			nTCPPort		:= TO_UINT(SlaveCom[SlaveNo]^.Port), 
			nUnitID			:= SlaveCom[SlaveNo]^.Address, 
			nQuantity		:= SlaveCom[SlaveNo]^.jobs[JobNo].Quantity, 
			nMBAddr			:= SlaveCom[SlaveNo]^.jobs[JobNo].startAddress, 
			cbLength		:= SlaveCom[SlaveNo]^.jobs[JobNo].Quantity, 
			pSrcAddr		:= ADR(SlaveCom[SlaveNo]^.Data), 
			bExecute		:= Execute, 
			tTimeout		:= , 
			bBusy			=> StartJob, 
			bError			=> Error, 
			nErrId			=> ErrorID);
	
	ELSIF 	SlaveCom[SlaveNo]^.Jobs[JobNo].FunctionCode = 16 THEN
		WriteRegs(
			sIPAddr			:= SlaveCom[SlaveNo]^.ipAddr, 
			nTCPPort		:= TO_UINT(SlaveCom[SlaveNo]^.Port), 
			nUnitID			:= SlaveCom[SlaveNo]^.Address, 
			nQuantity		:= SlaveCom[SlaveNo]^.jobs[JobNo].Quantity, 
			nMBAddr			:= SlaveCom[SlaveNo]^.jobs[JobNo].startAddress, 
			cbLength		:= SlaveCom[SlaveNo]^.jobs[JobNo].Quantity, 
			pSrcAddr		:= ADR(SlaveCom[SlaveNo]^.Data), 
			bExecute		:= Execute, 
			tTimeout		:= , 
			bBusy			=> StartJob, 
			bError			=> Error, 
			nErrId			=> ErrorID);
			
	ELSIF 	SlaveCom[SlaveNo]^.Jobs[JobNo].FunctionCode = 23 THEN
		// not implemented
(*		ReadWriteRegs(
			sIPAddr			:= SlaveCom[SlaveNo]^.ipAddr, 
			nTCPPort		:= SlaveCom[SlaveNo]^.Port, 
			nUnitID			:= SlaveCom[SlaveNo]^.Address, 
			nReadQuantity	:= SlaveCom[SlaveNo]^.jobs[JobNo].Quantity, 
			nMBReadAddr		:= SlaveCom[SlaveNo]^.jobs[JobNo].startAddress, 
			nWriteQuantity	:= , // missing
			nMBWriteAddr	:= , // missing
			cbDestLength	:= SlaveCom[SlaveNo]^.jobs[JobNo].Quantity, 
			pDestAddr		:= ADR(SlaveCom[SlaveNo]^.Data),
			cbSrcLength		:= , // missing
			pSrcAddr 		:= , // missing
			bExecute		:= Execute, 
			tTimeout		:= , 
			bBusy			=> StartJob, 
			bError			=> Error, 
			nErrId			=> ErrorID);	

*)			
	END_IF
END_METHOD

END_FUNCTION_BLOCK

// POUs/Connectivity/TF625x-Modbus/Master/TF6255-ModbusRtu/ModbusRtuMaster22B
{attribute 'no_check'}
// ModBus comunication master to multible slaves useing RTU protocol
// based on TF6255 - required lib: Tc2_ModbusRTU
FUNCTION_BLOCK ModbusRtuMaster22B
VAR CONSTANT
	MIN_SLAVE												:	INT := 1;
	MAX_SLAVE												:	INT := PARAM.MODBUS_MAX_SLAVES_OF_MASTER;
END_VAR
VAR_INPUT
	Enable													:	BOOL ; 			// FB will be processed as long as enable is TRUE 
	ResetTrig												:	BOOL ;			// The function block will be reset with a rising edge 
	SlaveCom												:	ARRAY[MIN_SLAVE..MAX_SLAVE] OF POINTER TO ModbusSlaveCom;
	Timestamp												:	DT;
END_VAR         	
VAR_OUTPUT      	
	Error													:	BOOL;			// Rising edge of Error informs that an error occurred during the execution of the Function Block 
	ErrorID													:	MODBUS_ERRORS;	// Error identification 
	ErrorText												:	STRING;
END_VAR
VAR
(* memory **************************************************)
	state 													:	INT := 0;
	JobNo													:	INT := 0;
	SlaveNo													:	INT := 0;
(* trigger *************************************************)

(* timer ***************************************************)

(* blocks **************************************************)
//	com														:	ModbusRtuMaster_PcCOM := (Timeout := DEFAULT_ADS_TIMEOUT);
	com														:	ModbusRtuMaster_KL6x22B := (Timeout := DEFAULT_ADS_TIMEOUT);
//	com														:	ModbusRtuMaster_KL6x5B := (Timeout := DEFAULT_ADS_TIMEOUT);
(* internal used variables *********************************)
	i,j,k													:	INT :=0;
END_VAR

(* ModBus RTU comunication to multible slaves 	JHue V1.0			*)
(* uncomment necessary master funktion block 						*)
(* use TC2_ModBusRTU.lib											*)
(********************************************************************)
	CASE state OF
	0:	(* Idle *)
		IF Enable 
		THEN
			k 												:=	0;
			JobNo  :=  SlaveNo								:=	1;
			state 											:=	10;
		END_IF

	10: 
		IF GetNextSlave() 
		THEN (* find Slave *)
			k 												:= 0;
			IF GetNextJob() 
			THEN (* find JobNo *)
				SlaveCom[SlaveNo]^.currentJobIdx 			:= JobNo;
				SlaveCom[SlaveNo]^.writeJobRequested 		:= SlaveCom[SlaveNo]^.Jobs[JobNo].FunctionCode >= 5;
				State 										:= SEL(SlaveCom[SlaveNo]^.writeJobRequested, 20, 15);
			END_IF
		ELSE
			state 											:=	0;
		END_IF
	
	15: (* wait for valid write date *)
		IF NOT SlaveCom[SlaveNo]^.writeJobRequested
		THEN
			SlaveCom[SlaveNo]^.Jobs[JobNo].Valid 			:= FALSE;
			state 											:= 20;
		END_IF

	20: (* start job *)	
		IF NOT StartJob(FALSE) // Busy
		THEN						
			state 											:= 30;
		END_IF

	30: (* wait for com cycle *)
		IF NOT StartJob(TRUE) THEN // Busy
			IF Error 
			THEN
				ErrorText									:= CONCAT('Error at SlaveNo: ',	CONCAT(INT_TO_STRING(SlaveNo), CONCAT(', JobNo: ', INT_TO_STRING(JobNo))));
				SlaveCom[SlaveNo]^.countBad 				:= SlaveCom[SlaveNo]^.countBad +1;
				state 										:= 98; 
			ELSE
				SlaveCom[SlaveNo]^.countGood 				:= SlaveCom[SlaveNo]^.countGood +1;
				SlaveCom[SlaveNo]^.Jobs[JobNo].Valid 		:= TRUE;
				SlaveCom[SlaveNo]^.Jobs[JobNo].TimeStamp 	:= Timestamp;
				JobNo 										:= JobNo + 1;
				state 										:= 10;	(* next job *)
			END_IF
			StartJob(FALSE);
		END_IF

	98: (* wait for quit *)
		IF ResetTrig THEN
			reset();
		END_IF

	END_CASE

METHOD PRIVATE getNextJob : Bool //Return value = TRUE if execution finished
VAR_INPUT
END_VAR
	
	WHILE SlaveCom[SlaveNo]^.Jobs[JobNo].FunctionCode = 0 DO
		JobNo 											:= JobNo + 1;
		IF JobNo > SlaveCom[SlaveNo]^.MAX_SLAVE_JOB THEN
			JobNo 										:= SlaveCom[SlaveNo]^.MIN_SLAVE_JOB;
			SlaveNo 									:= SlaveNo + 1;
			GetNextJob									:= FALSE;
			RETURN;
		END_IF
	END_WHILE
	GetNextJob											:= TRUE;
END_METHOD

METHOD PRIVATE getNextSlave : Bool //Return value = TRUE if execution finished
VAR_INPUT
END_VAR
	WHILE SlaveCom[SlaveNo] = 0 OR_ELSE NOT SlaveCom[SlaveNo]^.Enable DO
		SlaveNo 										:= SlaveNo + 1;
		IF SlaveNo > MAX_SLAVE 
		THEN
			k 											:= k + 1;
			SlaveNo 									:= MIN_SLAVE;
		ELSIF k = 2 
		THEN
			k 											:= 0;
			GetNextSlave								:= FALSE;
			RETURN;
		END_IF	
	END_WHILE
	GetNextSlave										:= TRUE;
END_METHOD

METHOD PUBLIC reset : BOOL //Return value = TRUE if execution finished
VAR_INPUT
END_VAR
IF State = 98 
THEN
	Error													:= FALSE;
	ErrorID													:= 0;
	ErrorText												:= '';
	state													:= 0;
END_IF
reset													:= TRUE;
END_METHOD

METHOD PRIVATE startJob : BOOL //Return value = TRUE if busy - TRUE as long as the job is busy
VAR_INPUT
	Execute							: BOOL;
END_VAR
(* ModbusCOM Baustein mit parametern antriggern *)
	IF 		SlaveCom[SlaveNo]^.Jobs[JobNo].FunctionCode = 1 THEN
		com.ReadCoils(
			UnitID			:= SlaveCom[SlaveNo]^.Address,					(*UnitID: Modbus Stationsadresse (1..247). Der Modbus-Slave antwortet nur, wenn er Telegramme mit seiner eigenen Stationsadresse empfängt. optional können hier auch Sammeladressen eingestellt werden um auf beliebige Anfragen zu antworten. Die Adresse 0 ist für Broadcast-Telegramme reserviert und somit keine gültige Stationsadresse.*)
			Quantity		:= SlaveCom[SlaveNo]^.jobs[JobNo].Quantity,		(*Quantity: Anzahl der zu lesenden oder zu schreibenden Datenworte bei Wort-orientierten Modbus-Funktionen. Bei Bit-orientierten Modbus-Funktionen gibt Quantity die Anzahl der Bits (Inputs oder Coils) an.*)
			MBAddr			:= SlaveCom[SlaveNo]^.jobs[JobNo].startAddress,	(*MBAddr: Modbus-Datenadresse, von der die Daten aus dem Endgerät (Slave) gelesen werden. Diese Adresse wird unverändert zum Slave übertragen und wird dort als Datenadresse interpretiert.*)
			cbLength		:= SlaveCom[SlaveNo]^.jobs[JobNo].Quantity, 	(*cbLength : Größe der verwendeten Datenvariable für Sende- oder Lese-Aktionen in Bytes. cbLength muss größer oder gleich der durch Quantity bestimmten übertragenen Datenmenge sein. Bei Wortzugriffen gilt z. B.: [cbLength >= Quantity * 2]. cbLength kann mit SIZEOF(ModbusDaten) berechnet werden.*)
			pMemoryAddr		:= ADR(SlaveCom[SlaveNo]^.Data),				(*pMemoryAddr: Speicheradresse in der SPS, die mit ADR(ModbusDaten) berechnet wird. Bei Leseaktionen werden die gelesenen Daten in der adressierten Variablen abgelegt. Bei Sende-Aktionen werden die Daten aus der adressierten Variablen zum Endgerät übertragen.*)
			Execute			:= Execute,
			Timeout			:= ,
			BUSY			=> StartJob,									(*Busy: Zeigt an, dass der Funktionsbaustein aktiv ist. Busy wird mit steigender Flanke an Execute TRUE und wird wieder FALSE nachdem die gestartete Aktion beendet ist. Es kann immer nur eine Aktion gleichzeitig aktiv sein.*)
			Error			=> Error,										(*Error: Zeigt an, dass bei der Bearbeitung einer Aktion ein Fehler aufgetreten ist*)
			ErrorId			=> ErrorID);									(*ErrorId: Zeigt eine Fehlernummer im Falle einer gestörten oder fehlerhaften Kommunikation an.*)	

	ELSIF 	SlaveCom[SlaveNo]^.Jobs[JobNo].FunctionCode = 3 THEN
		com.ReadRegs(
			UnitID			:= SlaveCom[SlaveNo]^.Address,		
			Quantity		:= SlaveCom[SlaveNo]^.jobs[JobNo].Quantity,
			MBAddr			:= SlaveCom[SlaveNo]^.jobs[JobNo].startAddress,
			cbLength		:= SlaveCom[SlaveNo]^.jobs[JobNo].Quantity * 2,
			pMemoryAddr		:= ADR(SlaveCom[SlaveNo]^.data),
			Execute			:= Execute,
			Timeout			:= ,
			BUSY			=> StartJob,
			Error			=> Error,
			ErrorId			=> ErrorID);
	
	ELSIF 	SlaveCom[SlaveNo]^.Jobs[JobNo].FunctionCode = 4 THEN
		com.ReadInputRegs(
			UnitID			:= SlaveCom[SlaveNo]^.Address,		
			Quantity		:= SlaveCom[SlaveNo]^.jobs[JobNo].Quantity,
			MBAddr			:= SlaveCom[SlaveNo]^.jobs[JobNo].startAddress,
			cbLength		:= SlaveCom[SlaveNo]^.jobs[JobNo].Quantity * 2,
			pMemoryAddr		:= ADR(SlaveCom[SlaveNo]^.data),
			Execute			:= Execute,
			Timeout			:= ,
			BUSY			=> StartJob,
			Error			=> Error,
			ErrorId			=> ErrorID);
	
	ELSIF 	SlaveCom[SlaveNo]^.Jobs[JobNo].FunctionCode = 5 THEN
		com.WriteSingleCoil(
			UnitID			:= SlaveCom[SlaveNo]^.Address,		
			Quantity		:= SlaveCom[SlaveNo]^.jobs[JobNo].Quantity,
			MBAddr			:= SlaveCom[SlaveNo]^.jobs[JobNo].startAddress,
			cbLength		:= SlaveCom[SlaveNo]^.jobs[JobNo].Quantity,
			pMemoryAddr		:= ADR(SlaveCom[SlaveNo]^.data),
			Execute			:= Execute,
			Timeout			:= ,
			BUSY			=> StartJob,
			Error			=> Error,
			ErrorId			=> ErrorID);
			
	ELSIF 	SlaveCom[SlaveNo]^.Jobs[JobNo].FunctionCode = 6 THEN
		com.WriteSingleRegister(
			UnitID			:= SlaveCom[SlaveNo]^.Address,		
			Quantity		:= SlaveCom[SlaveNo]^.jobs[JobNo].Quantity,
			MBAddr			:= SlaveCom[SlaveNo]^.jobs[JobNo].startAddress,
			cbLength		:= SlaveCom[SlaveNo]^.jobs[JobNo].Quantity,
			pMemoryAddr		:= ADR(SlaveCom[SlaveNo]^.data),
			Execute			:= Execute,
			Timeout			:= ,
			BUSY			=> StartJob,
			Error			=> Error,
			ErrorId			=> ErrorID);
		
	ELSIF 	SlaveCom[SlaveNo]^.Jobs[JobNo].FunctionCode = 8 THEN
		com.Diagnostics(
			UnitID			:= SlaveCom[SlaveNo]^.Address,		
			Quantity		:= SlaveCom[SlaveNo]^.jobs[JobNo].Quantity,
			MBAddr			:= SlaveCom[SlaveNo]^.jobs[JobNo].startAddress,
			cbLength		:= SlaveCom[SlaveNo]^.jobs[JobNo].Quantity,
			pMemoryAddr		:= ADR(SlaveCom[SlaveNo]^.data),
			Execute			:= Execute,
			Timeout			:= ,
			BUSY			=> StartJob,
			Error			=> Error,
			ErrorId			=> ErrorID);
		
	ELSIF 	SlaveCom[SlaveNo]^.Jobs[JobNo].FunctionCode = 15 THEN
		com.WriteMultipleCoils(
			UnitID			:= SlaveCom[SlaveNo]^.Address,		
			Quantity		:= SlaveCom[SlaveNo]^.jobs[JobNo].Quantity,
			MBAddr			:= SlaveCom[SlaveNo]^.jobs[JobNo].startAddress,
			cbLength		:= SlaveCom[SlaveNo]^.jobs[JobNo].Quantity,
			pMemoryAddr		:= ADR(SlaveCom[SlaveNo]^.data),
			Execute			:= Execute,
			Timeout			:= ,
			BUSY			=> StartJob,
			Error			=> Error,
			ErrorId			=> ErrorID);
	
	ELSIF 	SlaveCom[SlaveNo]^.Jobs[JobNo].FunctionCode = 16 THEN
		com.WriteRegs(
			UnitID			:= SlaveCom[SlaveNo]^.Address,		
			Quantity		:= SlaveCom[SlaveNo]^.jobs[JobNo].Quantity,
			MBAddr			:= SlaveCom[SlaveNo]^.jobs[JobNo].startAddress,
			cbLength		:= SlaveCom[SlaveNo]^.jobs[JobNo].Quantity,
			pMemoryAddr		:= ADR(SlaveCom[SlaveNo]^.data),
			Execute			:= Execute,
			Timeout			:= ,
			BUSY			=> StartJob,
			Error			=> Error,
			ErrorId			=> ErrorID);
			
	END_IF
END_METHOD

END_FUNCTION_BLOCK

// POUs/Connectivity/TF625x-Modbus/Master/TF6255-ModbusRtu/ModbusRtuMaster5B
{attribute 'no_check'}
// ModBus comunication master to multible slaves useing RTU protocol
// based on TF6255 - required lib: Tc2_ModbusRTU
FUNCTION_BLOCK ModbusRtuMaster5B
VAR CONSTANT
	MIN_SLAVE												:	INT := 1;
	MAX_SLAVE												:	INT := PARAM.MODBUS_MAX_SLAVES_OF_MASTER;
END_VAR
VAR_INPUT
	Enable													:	BOOL ; 			// FB will be processed as long as enable is TRUE 
	ResetTrig												:	BOOL ;			// The function block will be reset with a rising edge 
	SlaveCom												:	ARRAY[MIN_SLAVE..MAX_SLAVE] OF POINTER TO ModbusSlaveCom;
	Timestamp												:	DT;
END_VAR         	
VAR_OUTPUT      	
	Error													:	BOOL;			// Rising edge of Error informs that an error occurred during the execution of the Function Block 
	ErrorID													:	MODBUS_ERRORS;	// Error identification 
	ErrorText												:	STRING;
END_VAR
VAR
(* memory **************************************************)
	state 													:	INT := 0;
	JobNo													:	INT := 0;
	SlaveNo													:	INT := 0;
(* trigger *************************************************)

(* timer ***************************************************)

(* blocks **************************************************)
//	com														:	ModbusRtuMaster_PcCOM := (Timeout := DEFAULT_ADS_TIMEOUT);
//	com														:	ModbusRtuMaster_KL6x22B := (Timeout := DEFAULT_ADS_TIMEOUT);
	com														:	ModbusRtuMaster_KL6x5B := (Timeout := DEFAULT_ADS_TIMEOUT);
(* internal used variables *********************************)
	i,j,k													:	INT :=0;
END_VAR

(* ModBus RTU comunication to multible slaves 	JHue V1.0			*)
(* uncomment necessary master funktion block 						*)
(* use TC2_ModBusRTU.lib											*)
(********************************************************************)
	CASE state OF
	0:	(* Idle *)
		IF Enable 
		THEN
			k 												:=	0;
			JobNo  :=  SlaveNo								:=	1;
			state 											:=	10;
		END_IF

	10: 
		IF GetNextSlave() 
		THEN (* find Slave *)
			k 												:= 0;
			IF GetNextJob() 
			THEN (* find JobNo *)
				SlaveCom[SlaveNo]^.currentJobIdx 			:= JobNo;
				SlaveCom[SlaveNo]^.writeJobRequested 		:= SlaveCom[SlaveNo]^.Jobs[JobNo].FunctionCode >= 5;
				State 										:= SEL(SlaveCom[SlaveNo]^.writeJobRequested, 20, 15);
			END_IF
		ELSE
			state 											:=	0;
		END_IF
	
	15: (* wait for valid write date *)
		IF NOT SlaveCom[SlaveNo]^.writeJobRequested
		THEN
			SlaveCom[SlaveNo]^.Jobs[JobNo].Valid 			:= FALSE;
			state 											:= 20;
		END_IF

	20: (* start job *)	
		IF NOT StartJob(FALSE) // Busy
		THEN						
			state 											:= 30;
		END_IF

	30: (* wait for com cycle *)
		IF NOT StartJob(TRUE) THEN // Busy
			IF Error 
			THEN
				ErrorText									:= CONCAT('Error at SlaveNo: ',	CONCAT(INT_TO_STRING(SlaveNo), CONCAT(', JobNo: ', INT_TO_STRING(JobNo))));
				SlaveCom[SlaveNo]^.countBad 				:= SlaveCom[SlaveNo]^.countBad +1;
				state 										:= 98; 
			ELSE
				SlaveCom[SlaveNo]^.countGood 				:= SlaveCom[SlaveNo]^.countGood +1;
				SlaveCom[SlaveNo]^.Jobs[JobNo].Valid 		:= TRUE;
				SlaveCom[SlaveNo]^.Jobs[JobNo].TimeStamp 	:= Timestamp;
				JobNo 										:= JobNo + 1;
				state 										:= 10;	(* next job *)
			END_IF
			StartJob(FALSE);
		END_IF

	98: (* wait for quit *)
		IF ResetTrig THEN
			reset();
		END_IF

	END_CASE

METHOD PRIVATE getNextJob : Bool
VAR_INPUT
END_VAR
	
	WHILE SlaveCom[SlaveNo]^.Jobs[JobNo].FunctionCode = 0 DO
		JobNo 											:= JobNo + 1;
		IF JobNo > SlaveCom[SlaveNo]^.MAX_SLAVE_JOB THEN
			JobNo 										:= SlaveCom[SlaveNo]^.MIN_SLAVE_JOB;
			SlaveNo 									:= SlaveNo + 1;
			GetNextJob									:= FALSE;
			RETURN;
		END_IF
	END_WHILE
	GetNextJob											:= TRUE;
END_METHOD

METHOD PRIVATE getNextSlave : Bool
VAR_INPUT
END_VAR
	WHILE SlaveCom[SlaveNo] = 0 OR_ELSE NOT SlaveCom[SlaveNo]^.Enable DO
		SlaveNo 										:= SlaveNo + 1;
		IF SlaveNo > MAX_SLAVE 
		THEN
			k 											:= k + 1;
			SlaveNo 									:= MIN_SLAVE;
		ELSIF k = 2 
		THEN
			k 											:= 0;
			GetNextSlave								:= FALSE;
			RETURN;
		END_IF	
	END_WHILE
	GetNextSlave										:= TRUE;
END_METHOD

METHOD PUBLIC reset : booL //Return value = TRUE if execution finished
VAR_INPUT
END_VAR
IF State = 98 
THEN
	Error													:= FALSE;
	ErrorID													:= 0;
	ErrorText												:= '';
	state													:= 0;
END_IF
reset													:= TRUE;
END_METHOD

METHOD PRIVATE startJob : BOOL //Return value = TRUE if busy - TRUE as long as the job is busy
VAR_INPUT
	Execute							: BOOL;
END_VAR
(* ModbusCOM Baustein mit parametern antriggern *)
	IF 		SlaveCom[SlaveNo]^.Jobs[JobNo].FunctionCode = 1 THEN
		com.ReadCoils(
			UnitID			:= SlaveCom[SlaveNo]^.Address,				(*UnitID: Modbus Stationsadresse (1..247). Der Modbus-Slave antwortet nur, wenn er Telegramme mit seiner eigenen Stationsadresse empfängt. optional können hier auch Sammeladressen eingestellt werden um auf beliebige Anfragen zu antworten. Die Adresse 0 ist für Broadcast-Telegramme reserviert und somit keine gültige Stationsadresse.*)
			Quantity		:= SlaveCom[SlaveNo]^.jobs[JobNo].Quantity,		(*Quantity: Anzahl der zu lesenden oder zu schreibenden Datenworte bei Wort-orientierten Modbus-Funktionen. Bei Bit-orientierten Modbus-Funktionen gibt Quantity die Anzahl der Bits (Inputs oder Coils) an.*)
			MBAddr			:= SlaveCom[SlaveNo]^.jobs[JobNo].startAddress,	(*MBAddr: Modbus-Datenadresse, von der die Daten aus dem Endgerät (Slave) gelesen werden. Diese Adresse wird unverändert zum Slave übertragen und wird dort als Datenadresse interpretiert.*)
			cbLength		:= SlaveCom[SlaveNo]^.jobs[JobNo].Quantity, 	(*cbLength : Größe der verwendeten Datenvariable für Sende- oder Lese-Aktionen in Bytes. cbLength muss größer oder gleich der durch Quantity bestimmten übertragenen Datenmenge sein. Bei Wortzugriffen gilt z. B.: [cbLength >= Quantity * 2]. cbLength kann mit SIZEOF(ModbusDaten) berechnet werden.*)
			pMemoryAddr		:= ADR(SlaveCom[SlaveNo]^.Data),				(*pMemoryAddr: Speicheradresse in der SPS, die mit ADR(ModbusDaten) berechnet wird. Bei Leseaktionen werden die gelesenen Daten in der adressierten Variablen abgelegt. Bei Sende-Aktionen werden die Daten aus der adressierten Variablen zum Endgerät übertragen.*)
			Execute			:= Execute,
			Timeout			:= ,
			BUSY			=> StartJob,									(*Busy: Zeigt an, dass der Funktionsbaustein aktiv ist. Busy wird mit steigender Flanke an Execute TRUE und wird wieder FALSE nachdem die gestartete Aktion beendet ist. Es kann immer nur eine Aktion gleichzeitig aktiv sein.*)
			Error			=> Error,										(*Error: Zeigt an, dass bei der Bearbeitung einer Aktion ein Fehler aufgetreten ist*)
			ErrorId			=> ErrorID);									(*ErrorId: Zeigt eine Fehlernummer im Falle einer gestörten oder fehlerhaften Kommunikation an.*)	
	
	ELSIF 	SlaveCom[SlaveNo]^.Jobs[JobNo].FunctionCode = 3 THEN
		com.ReadRegs(
			UnitID			:= SlaveCom[SlaveNo]^.Address,		
			Quantity		:= SlaveCom[SlaveNo]^.jobs[JobNo].Quantity,
			MBAddr			:= SlaveCom[SlaveNo]^.jobs[JobNo].startAddress,
			cbLength		:= SlaveCom[SlaveNo]^.jobs[JobNo].Quantity * 2,
			pMemoryAddr		:= ADR(SlaveCom[SlaveNo]^.data),
			Execute			:= Execute,
			Timeout			:= ,
			BUSY			=> StartJob,
			Error			=> Error,
			ErrorId			=> ErrorID);
	
	ELSIF 	SlaveCom[SlaveNo]^.Jobs[JobNo].FunctionCode = 4 THEN
		com.ReadInputRegs(
			UnitID			:= SlaveCom[SlaveNo]^.Address,		
			Quantity		:= SlaveCom[SlaveNo]^.jobs[JobNo].Quantity,
			MBAddr			:= SlaveCom[SlaveNo]^.jobs[JobNo].startAddress,
			cbLength		:= SlaveCom[SlaveNo]^.jobs[JobNo].Quantity * 2,
			pMemoryAddr		:= ADR(SlaveCom[SlaveNo]^.data),
			Execute			:= Execute,
			Timeout			:= ,
			BUSY			=> StartJob,
			Error			=> Error,
			ErrorId			=> ErrorID);
	
	ELSIF 	SlaveCom[SlaveNo]^.Jobs[JobNo].FunctionCode = 5 THEN
		com.WriteSingleCoil(
			UnitID			:= SlaveCom[SlaveNo]^.Address,		
			Quantity		:= SlaveCom[SlaveNo]^.jobs[JobNo].Quantity,
			MBAddr			:= SlaveCom[SlaveNo]^.jobs[JobNo].startAddress,
			cbLength		:= SlaveCom[SlaveNo]^.jobs[JobNo].Quantity,
			pMemoryAddr		:= ADR(SlaveCom[SlaveNo]^.data),
			Execute			:= Execute,
			Timeout			:= ,
			BUSY			=> StartJob,
			Error			=> Error,
			ErrorId			=> ErrorID);
		
	ELSIF 	SlaveCom[SlaveNo]^.Jobs[JobNo].FunctionCode = 6 THEN
		com.WriteSingleRegister(
			UnitID			:= SlaveCom[SlaveNo]^.Address,		
			Quantity		:= SlaveCom[SlaveNo]^.jobs[JobNo].Quantity,
			MBAddr			:= SlaveCom[SlaveNo]^.jobs[JobNo].startAddress,
			cbLength		:= SlaveCom[SlaveNo]^.jobs[JobNo].Quantity,
			pMemoryAddr		:= ADR(SlaveCom[SlaveNo]^.data),
			Execute			:= Execute,
			Timeout			:= ,
			BUSY			=> StartJob,
			Error			=> Error,
			ErrorId			=> ErrorID);
			
	ELSIF 	SlaveCom[SlaveNo]^.Jobs[JobNo].FunctionCode = 8 THEN
		com.Diagnostics(
			UnitID			:= SlaveCom[SlaveNo]^.Address,		
			Quantity		:= SlaveCom[SlaveNo]^.jobs[JobNo].Quantity,
			MBAddr			:= SlaveCom[SlaveNo]^.jobs[JobNo].startAddress,
			cbLength		:= SlaveCom[SlaveNo]^.jobs[JobNo].Quantity,
			pMemoryAddr		:= ADR(SlaveCom[SlaveNo]^.data),
			Execute			:= Execute,
			Timeout			:= ,
			BUSY			=> StartJob,
			Error			=> Error,
			ErrorId			=> ErrorID);
	
	ELSIF 	SlaveCom[SlaveNo]^.Jobs[JobNo].FunctionCode = 15 THEN
		com.WriteMultipleCoils(
			UnitID			:= SlaveCom[SlaveNo]^.Address,		
			Quantity		:= SlaveCom[SlaveNo]^.jobs[JobNo].Quantity,
			MBAddr			:= SlaveCom[SlaveNo]^.jobs[JobNo].startAddress,
			cbLength		:= SlaveCom[SlaveNo]^.jobs[JobNo].Quantity,
			pMemoryAddr		:= ADR(SlaveCom[SlaveNo]^.data),
			Execute			:= Execute,
			Timeout			:= ,
			BUSY			=> StartJob,
			Error			=> Error,
			ErrorId			=> ErrorID);
	
	ELSIF 	SlaveCom[SlaveNo]^.Jobs[JobNo].FunctionCode = 16 THEN
		com.WriteRegs(
			UnitID			:= SlaveCom[SlaveNo]^.Address,		
			Quantity		:= SlaveCom[SlaveNo]^.jobs[JobNo].Quantity,
			MBAddr			:= SlaveCom[SlaveNo]^.jobs[JobNo].startAddress,
			cbLength		:= SlaveCom[SlaveNo]^.jobs[JobNo].Quantity,
			pMemoryAddr		:= ADR(SlaveCom[SlaveNo]^.data),
			Execute			:= Execute,
			Timeout			:= ,
			BUSY			=> StartJob,
			Error			=> Error,
			ErrorId			=> ErrorID);	
	END_IF
END_METHOD

END_FUNCTION_BLOCK

// POUs/Connectivity/TF625x-Modbus/Master/TF6255-ModbusRtu/ModbusRtuMasterPC
{attribute 'no_check'}
// ModBus comunication master to multible slaves useing RTU protocol
// based on TF6255 - required lib: Tc2_ModbusRTU
FUNCTION_BLOCK ModbusRtuMasterPC
VAR CONSTANT
	MIN_SLAVE												:	INT := 1;
	MAX_SLAVE												:	INT := PARAM.MODBUS_MAX_SLAVES_OF_MASTER;
END_VAR
VAR_INPUT
	Enable													:	BOOL; 			// FB will be processed as long as enable is TRUE 
	ResetTrig												:	BOOL;			// The function block will be reset with a rising edge 
	SlaveCom												:	ARRAY[MIN_SLAVE..MAX_SLAVE] OF POINTER TO ModbusSlaveCom;
	Timestamp												:	DT;
END_VAR         	
VAR_OUTPUT      	
	Error													:	BOOL;			// Rising edge of Error informs that an error occurred during the execution of the Function Block 
	ErrorID													:	MODBUS_ERRORS;	// Error identification 
	ErrorText												:	STRING;
END_VAR
VAR
(* memory **************************************************)
	state 													:	INT := 0;
	JobNo													:	INT := 0;
	SlaveNo													:	INT := 0;
(* trigger *************************************************)

(* timer ***************************************************)

(* blocks **************************************************)
	com														:	ModbusRtuMaster_PcCOM := (Timeout := DEFAULT_ADS_TIMEOUT);
//	com														:	ModbusRtuMaster_KL6x22B := (Timeout := DEFAULT_ADS_TIMEOUT);
//	com														:	ModbusRtuMaster_KL6x5B := (Timeout := DEFAULT_ADS_TIMEOUT);
(* internal used variables *********************************)
	i,j,k													:	INT :=0;

END_VAR

(* ModBus RTU comunication to multible slaves 	JHue V1.0			*)
(* uncomment necessary master funktion block 						*)
(* use TC2_ModBusRTU.lib											*)
(********************************************************************)

	CASE state OF
	0:	(* Idle *)
		IF Enable 
		THEN
			k 												:=	0;
			JobNo  :=  SlaveNo								:=	1;
			state 											:=	10;
		END_IF

	10: 
		IF GetNextSlave() 
		THEN (* find Slave *)
			k 												:= 0;
			IF GetNextJob() 
			THEN (* find JobNo *)
				SlaveCom[SlaveNo]^.currentJobIdx 			:= JobNo;
				SlaveCom[SlaveNo]^.writeJobRequested 		:= SlaveCom[SlaveNo]^.Jobs[JobNo].FunctionCode >= 5;
				State 										:= SEL(SlaveCom[SlaveNo]^.writeJobRequested, 20, 15);
			END_IF
		ELSE
			state 											:=	0;
		END_IF
	
	15: (* wait for valid write date *)
		IF NOT SlaveCom[SlaveNo]^.writeJobRequested
		THEN
			SlaveCom[SlaveNo]^.Jobs[JobNo].Valid 			:= FALSE;
			state 											:= 0;
		END_IF

	20: (* start job *)	
		IF NOT StartJob(FALSE) // Busy
		THEN						
			state 											:= 30;
		END_IF

	30: (* wait for com cycle *)
		IF NOT StartJob(TRUE) THEN // Busy
			IF Error 
			THEN
				ErrorText									:= CONCAT('Error at SlaveNo: ',	CONCAT(INT_TO_STRING(SlaveNo), CONCAT(', JobNo: ', INT_TO_STRING(JobNo))));
				SlaveCom[SlaveNo]^.countBad 				:= SlaveCom[SlaveNo]^.countBad +1;
				state 										:= 98; 
			ELSE
				SlaveCom[SlaveNo]^.countGood 				:= SlaveCom[SlaveNo]^.countGood +1;
				SlaveCom[SlaveNo]^.Jobs[JobNo].Valid 		:= TRUE;
				SlaveCom[SlaveNo]^.Jobs[JobNo].TimeStamp 	:= Timestamp;
				JobNo 										:= JobNo + 1;
				state 										:= 10;	(* next job *)
			END_IF
			StartJob(FALSE);
		END_IF

	98: (* wait for quit *)
		IF ResetTrig THEN
			reset();
		END_IF

	END_CASE

METHOD PRIVATE getNextJob : Bool
VAR_INPUT
END_VAR
	
	WHILE SlaveCom[SlaveNo]^.Jobs[JobNo].FunctionCode = 0 DO
		JobNo 											:= JobNo + 1;
		IF JobNo > SlaveCom[SlaveNo]^.MAX_SLAVE_JOB THEN
			JobNo 										:= SlaveCom[SlaveNo]^.MIN_SLAVE_JOB;
			SlaveNo 									:= SlaveNo + 1;
			GetNextJob									:= FALSE;
			RETURN;
		END_IF
	END_WHILE
	GetNextJob											:= TRUE;
END_METHOD

METHOD PRIVATE getNextSlave : Bool
VAR_INPUT
END_VAR
	WHILE SlaveCom[SlaveNo] = 0 or_else not SlaveCom[SlaveNo]^.Enable DO
		SlaveNo 										:= SlaveNo + 1;
		IF SlaveNo > MAX_SLAVE 
		THEN
			k 											:= k + 1;
			SlaveNo 									:= MIN_SLAVE;
		ELSIF k = 2 
		THEN
			k 											:= 0;
			GetNextSlave								:= FALSE;
			RETURN;
		END_IF	
	END_WHILE
	GetNextSlave										:= TRUE;
END_METHOD

METHOD PUBLIC reset : BOOL //Return value = TRUE if execution finished
VAR_INPUT
END_VAR
IF State = 98 
THEN
	Error													:= FALSE;
	ErrorID													:= 0;
	ErrorText												:= '';
	state													:= 0;
END_IF
reset													:= TRUE;
END_METHOD

METHOD PRIVATE startJob : BOOL //Return value = TRUE if busy - TRUE as long as the job is busy
VAR_INPUT
	Execute							: BOOL;
END_VAR
(* ModbusCOM Baustein mit parametern antriggern *)
	IF 		SlaveCom[SlaveNo]^.Jobs[JobNo].FunctionCode = 1 THEN
		com.ReadCoils(
			UnitID			:= SlaveCom[SlaveNo]^.Address,				(*UnitID: Modbus Stationsadresse (1..247). Der Modbus-Slave antwortet nur, wenn er Telegramme mit seiner eigenen Stationsadresse empfängt. optional können hier auch Sammeladressen eingestellt werden um auf beliebige Anfragen zu antworten. Die Adresse 0 ist für Broadcast-Telegramme reserviert und somit keine gültige Stationsadresse.*)
			Quantity		:= SlaveCom[SlaveNo]^.jobs[JobNo].Quantity,		(*Quantity: Anzahl der zu lesenden oder zu schreibenden Datenworte bei Wort-orientierten Modbus-Funktionen. Bei Bit-orientierten Modbus-Funktionen gibt Quantity die Anzahl der Bits (Inputs oder Coils) an.*)
			MBAddr			:= SlaveCom[SlaveNo]^.jobs[JobNo].startAddress,	(*MBAddr: Modbus-Datenadresse, von der die Daten aus dem Endgerät (Slave) gelesen werden. Diese Adresse wird unverändert zum Slave übertragen und wird dort als Datenadresse interpretiert.*)
			cbLength		:= SlaveCom[SlaveNo]^.jobs[JobNo].Quantity, 	(*cbLength : Größe der verwendeten Datenvariable für Sende- oder Lese-Aktionen in Bytes. cbLength muss größer oder gleich der durch Quantity bestimmten übertragenen Datenmenge sein. Bei Wortzugriffen gilt z. B.: [cbLength >= Quantity * 2]. cbLength kann mit SIZEOF(ModbusDaten) berechnet werden.*)
			pMemoryAddr		:= ADR(SlaveCom[SlaveNo]^.Data),				(*pMemoryAddr: Speicheradresse in der SPS, die mit ADR(ModbusDaten) berechnet wird. Bei Leseaktionen werden die gelesenen Daten in der adressierten Variablen abgelegt. Bei Sende-Aktionen werden die Daten aus der adressierten Variablen zum Endgerät übertragen.*)
			Execute			:= Execute,
			Timeout			:= ,
			BUSY			=> StartJob,									(*Busy: Zeigt an, dass der Funktionsbaustein aktiv ist. Busy wird mit steigender Flanke an Execute TRUE und wird wieder FALSE nachdem die gestartete Aktion beendet ist. Es kann immer nur eine Aktion gleichzeitig aktiv sein.*)
			Error			=> Error,										(*Error: Zeigt an, dass bei der Bearbeitung einer Aktion ein Fehler aufgetreten ist*)
			ErrorId			=> ErrorID);									(*ErrorId: Zeigt eine Fehlernummer im Falle einer gestörten oder fehlerhaften Kommunikation an.*)	
	
	ELSIF 	SlaveCom[SlaveNo]^.Jobs[JobNo].FunctionCode = 3 THEN
		com.ReadRegs(
			UnitID			:= SlaveCom[SlaveNo]^.Address,		
			Quantity		:= SlaveCom[SlaveNo]^.jobs[JobNo].Quantity,
			MBAddr			:= SlaveCom[SlaveNo]^.jobs[JobNo].startAddress,
			cbLength		:= SlaveCom[SlaveNo]^.jobs[JobNo].Quantity * 2,
			pMemoryAddr		:= ADR(SlaveCom[SlaveNo]^.data),
			Execute			:= Execute,
			Timeout			:= ,
			BUSY			=> StartJob,
			Error			=> Error,
			ErrorId			=> ErrorID);
	
	ELSIF 	SlaveCom[SlaveNo]^.Jobs[JobNo].FunctionCode = 4 THEN
		com.ReadInputRegs(
			UnitID			:= SlaveCom[SlaveNo]^.Address,		
			Quantity		:= SlaveCom[SlaveNo]^.jobs[JobNo].Quantity,
			MBAddr			:= SlaveCom[SlaveNo]^.jobs[JobNo].startAddress,
			cbLength		:= SlaveCom[SlaveNo]^.jobs[JobNo].Quantity * 2,
			pMemoryAddr		:= ADR(SlaveCom[SlaveNo]^.data),
			Execute			:= Execute,
			Timeout			:= ,
			BUSY			=> StartJob,
			Error			=> Error,
			ErrorId			=> ErrorID);
	
	ELSIF 	SlaveCom[SlaveNo]^.Jobs[JobNo].FunctionCode = 5 THEN
		com.WriteSingleCoil(
			UnitID			:= SlaveCom[SlaveNo]^.Address,		
			Quantity		:= SlaveCom[SlaveNo]^.jobs[JobNo].Quantity,
			MBAddr			:= SlaveCom[SlaveNo]^.jobs[JobNo].startAddress,
			cbLength		:= SlaveCom[SlaveNo]^.jobs[JobNo].Quantity,
			pMemoryAddr		:= ADR(SlaveCom[SlaveNo]^.data),
			Execute			:= Execute,
			Timeout			:= ,
			BUSY			=> StartJob,
			Error			=> Error,
			ErrorId			=> ErrorID);
			
	ELSIF 	SlaveCom[SlaveNo]^.Jobs[JobNo].FunctionCode = 6 THEN
		com.WriteSingleRegister(
			UnitID			:= SlaveCom[SlaveNo]^.Address,		
			Quantity		:= SlaveCom[SlaveNo]^.jobs[JobNo].Quantity,
			MBAddr			:= SlaveCom[SlaveNo]^.jobs[JobNo].startAddress,
			cbLength		:= SlaveCom[SlaveNo]^.jobs[JobNo].Quantity,
			pMemoryAddr		:= ADR(SlaveCom[SlaveNo]^.data),
			Execute			:= Execute,
			Timeout			:= ,
			BUSY			=> StartJob,
			Error			=> Error,
			ErrorId			=> ErrorID);
		
	ELSIF 	SlaveCom[SlaveNo]^.Jobs[JobNo].FunctionCode = 8 THEN
		com.Diagnostics(
			UnitID			:= SlaveCom[SlaveNo]^.Address,		
			Quantity		:= SlaveCom[SlaveNo]^.jobs[JobNo].Quantity,
			MBAddr			:= SlaveCom[SlaveNo]^.jobs[JobNo].startAddress,
			cbLength		:= SlaveCom[SlaveNo]^.jobs[JobNo].Quantity,
			pMemoryAddr		:= ADR(SlaveCom[SlaveNo]^.data),
			Execute			:= Execute,
			Timeout			:= ,
			BUSY			=> StartJob,
			Error			=> Error,
			ErrorId			=> ErrorID);
	
	ELSIF 	SlaveCom[SlaveNo]^.Jobs[JobNo].FunctionCode = 15 THEN
		com.WriteMultipleCoils(
			UnitID			:= SlaveCom[SlaveNo]^.Address,		
			Quantity		:= SlaveCom[SlaveNo]^.jobs[JobNo].Quantity,
			MBAddr			:= SlaveCom[SlaveNo]^.jobs[JobNo].startAddress,
			cbLength		:= SlaveCom[SlaveNo]^.jobs[JobNo].Quantity,
			pMemoryAddr		:= ADR(SlaveCom[SlaveNo]^.data),
			Execute			:= Execute,
			Timeout			:= ,
			BUSY			=> StartJob,
			Error			=> Error,
			ErrorId			=> ErrorID);
	
	ELSIF 	SlaveCom[SlaveNo]^.Jobs[JobNo].FunctionCode = 16 THEN
		com.WriteRegs(
			UnitID			:= SlaveCom[SlaveNo]^.Address,		
			Quantity		:= SlaveCom[SlaveNo]^.jobs[JobNo].Quantity,
			MBAddr			:= SlaveCom[SlaveNo]^.jobs[JobNo].startAddress,
			cbLength		:= SlaveCom[SlaveNo]^.jobs[JobNo].Quantity,
			pMemoryAddr		:= ADR(SlaveCom[SlaveNo]^.data),
			Execute			:= Execute,
			Timeout			:= ,
			BUSY			=> StartJob,
			Error			=> Error,
			ErrorId			=> ErrorID);	
	END_IF
END_METHOD

END_FUNCTION_BLOCK

// POUs/Connectivity/TF625x-Modbus/Slave/ModbusSlaveBase
{attribute 'no_check'}
// Modbus SlaveRoot 
// This Funktionblock represents a root structure for a Modbus slave to communicate with all Modbus masters of Engineering Toolbox 
// inherit this POU into "your" Modbus device POU
// declare "your" Data POU for your Modbus Device
// overload methodes evaluation, initJobs and prepareWriteData as private and edit inbetween the marks
// call methode Run to start communication.
// based on TF625x Modbus communication
FUNCTION_BLOCK ModbusSlaveBase      
VAR_INPUT
	IpAddr													:	T_IPv4Addr := '127.0.0.1';	// use only for TCP and UDP or ''
	Port 													:	UDINT;			// use only for TCP			or 0
	Address													:	BYTE := 0;		//Modbus RTU addres
//	Data													:	MyModbusDeviceData;	
END_VAR            							
VAR_OUTPUT
	ModBusCom												:	ModbusSlaveCom; //Master-Slave Handshake object
	Valid													:	BOOL; 		//	data valid 
	TimeStamp												:	DT;			//	timestamp of last refresh 
	CountGood												:	DWORD := 0;	//	counter for successful data transmission 
	CountBad												:	DWORD := 0;	//	counter for failed data transmission
	NoOfJobs												:	INT;		//	no of active jobs
END_VAR
VAR
(* memory **************************************************)
	state													:	INT;						
(* trigger *************************************************)

(* timer ***************************************************)

(* blocks **************************************************)

(* internal used variables *********************************)
	i,j,k													:	INT :=0;	
END_VAR

;

METHOD PROTECTED evaluation : BOOL //Result needs to be TRUE if data are evaluated
VAR_INPUT
	CurrentJobIdx						: INT;
END_VAR
// copy and edit the code only between the marks to evaluate read data
	
	CASE currentJobIdx OF
	0: evaluation											:= TRUE;
	// **********************************************************		
	// Modify start *********************************************	
	1:	// evaluation of job 1 
		// Data.Var_a										:= ModBusCom.Data[1];
		// MEMCPY(ADR(Data.Var_b), ADR(ModBusCom.Data[1]),SIZEOF(Data.Var_b));
			// HOST_TO_BE16(Data.Var_b);		
		// MEMCPY(ADR(Data.Var_c), ADR(ModBusCom.Data[2]),SIZEOF(Data.Var_c));
			// HOST_TO_BE32(Data.Var_c);				
		//evaluation										:= TRUE;
	2:	// evaluation of job 2 
		// MEMCPY(ADR(Data.Var_d), ADR(ModBusCom.Data[1]),SIZEOF(Data.Var_a));
		// Data.Var_e										:=	DWORD_TO_REAL_EX(	ADR(ModBusCom.Data[	5	]));
		// Data.Var_f										:=	DWORD_TO_REAL_EX(	ADR(ModBusCom.Data[	9	]));	
		//evaluation										:= TRUE;	                                                
	3: 	// evaluation of job 3                              
		// Data.Var_g										:=	TO_INT(					ModBusCom.Data[	1	]);	
		// Data.Var_h										:=	TO_INT(					ModBusCom.Data[	3	]);
		// Data.Var_i										:=	TO_INT(					ModBusCom.Data[	5	]);
		//evaluation										:= TRUE;																					
	4:	// write job, no evaluation 	
		//evaluation										:= TRUE;
	// Modify end ***********************************************
	// **********************************************************
	ELSE
		;
	END_CASE
END_METHOD

METHOD PROTECTED initJobs : BOOL //Result needs to be TRUE for every valid JobIdx 
VAR_INPUT
	JobIdx													:	INT;
END_VAR
(********** Modbus slave jobs *********************)
	
// HINT: The register number is in accordance with the Modbus specification always less 1.
	CASE JobIdx OF
	0:initJobs												:= TRUE;
// **********************************************************		
// Modify start *********************************************
	1: // read job 
//		ModBusCom.Jobs[JobIdx].FunctionCode 				:=   3		;
//		ModBusCom.Jobs[JobIdx].startAddress					:=   499	;	(* first read-address -1 *)
//		ModBusCom.Jobs[JobIdx].Quantity 					:=   14		;	(* no of read words *)
//		initJobs											:= TRUE;
		                                    				
	2:	// read job                         				
//		ModBusCom.Jobs[JobIdx].FunctionCode 				:=   3		;
//		ModBusCom.Jobs[JobIdx].startAddress					:=  40000	;	(* first read-address -1 *)
//		ModBusCom.Jobs[JobIdx].Quantity 					:=   120	;	(* no of read words *)
//		initJobs											:= TRUE;
	3:	// read job                         				
//		ModBusCom.Jobs[JobIdx].FunctionCode 				:=   3		;
//		ModBusCom.Jobs[JobIdx].startAddress					:=  40120	;	(* first read-address -1 *)
//		ModBusCom.Jobs[JobIdx].Quantity 					:=   20		;	(* no of read words *)
//		initJobs											:= TRUE;
	4:	// write job                        				
//		ModBusCom.Jobs[JobIdx].FunctionCode 				:=   5		;
//		ModBusCom.Jobs[JobIdx].startAddress					:=   112	;	(* first read-address*)
//		ModBusCom.Jobs[JobIdx].Quantity 					:=   1		;	(* no of write words *)
//		initJobs											:= TRUE;
// Modify end ***********************************************
// **********************************************************	

	ELSE	
		;
	END_CASE
END_METHOD

METHOD PROTECTED prepareWriteData : BOOL	//Result needs to be TRUE for every valid write JobIdx
VAR_INPUT
	CurrentJobIdx						: INT;
END_VAR
// copy and edit the code only between the marks to prepare necessary write data
	CASE currentJobIdx OF	
	0:prepareWriteData										:= TRUE;
	// **********************************************************		
	// Modify start *********************************************
	1:	// no write data in this job
		
	2:	// no write data in this job
											
	3:  // no write data in this job
	
	4:	//Copy write job data to com object
		// ModBusCom.Data[	1	]							:=	Data.SET_Var_j;
		// prepareWriteData									:= TRUE; //Set to true:              			
	// Modify end ***********************************************
	// **********************************************************		
	ELSE
		;
	END_CASE
END_METHOD

METHOD FINAL run : BOOL // returns TRUE if one job is finished
VAR_INPUT
	Enable													:	BOOL;
END_VAR
	(* Modbus slave logic 									*)
	(********************************************************)
	
(* Sequence ****************************************************************)
CASE state OF 
//Wait for start slave 
0: 
	IF Enable 
	THEN
		ModBusCom.Enable									:= Enable;
		ModBusCom.Address 									:= Address;
		ModBusCom.IpAddr	 								:= IpAddr;
		ModBusCom.Port	 									:= Port;
		ModBusCom.countBad 		:= ModBusCom.countGood		:= 0;
		ModBusCom.noOfJobs 									:= 0;
		
		//Run loop to init every single job		
		FOR i:= ModBusCom.MIN_SLAVE_JOB TO ModBusCom.MAX_SLAVE_JOB DO
			ModBusCom.Jobs[i].Init();
			IF initJobs(JobIdx := i)
			THEN
				noOfJobs									:= i;
			ELSE
				EXIT;
			END_IF
		END_FOR

		ModBusCom.DeleteData();
		ModBusCom.noOfJobs									:= noOfJobs;
	
		state												:= 1;
	END_IF

//Read/write slave data is active
1: 
	//Init write data if requesed by master
	IF ModBusCom.writeJobRequested 
	THEN //
		ModBusCom.DeleteData();
		prepareWriteData(currentJobIdx := ModBusCom.currentJobIdx);
		ModBusCom.writeJobRequested 						:= FALSE;
	END_IF
	
	//Evaluation of job result
	IF ModBusCom.Jobs[ModBusCom.currentJobIdx].Valid //Valid is set by master
	THEN	
		Valid 												:= FALSE; //Slave data not valid
		evaluation(CurrentJobIdx := ModBusCom.currentJobIdx);	
				
		countBad 											:= ModBusCom.countBad;
		countGood 											:= ModBusCom.countGood;
		TimeStamp 											:= ModBusCom.Jobs[ModBusCom.currentJobIdx].TimeStamp;
		ModBusCom.Jobs[ModBusCom.currentJobIdx].Valid 		:= FALSE;
		ModBusCom.DeleteData();                                 
		Valid 												:= TRUE; //Slave data valid
		run													:= TRUE;
	ELSE
		run													:= FALSE;
	END_IF
	
	state													:= SEL(Enable, 0, state);
	ModBusCom.Enable										:= Enable;	
END_CASE
END_METHOD

END_FUNCTION_BLOCK

// POUs/Connectivity/TF6310-TcpServer/DeviceCom/TCPDeviceCom_SendRecBytes
//FB sends a "command" out and waits for response of the connected device (handshake mode)
//By setting pDest = 0 the FB will turn into only send mode and with pSrc = 0 into only receive mode (ClrComBuffer will be ignored)
FUNCTION_BLOCK TCPDeviceCom_SendRecBytes EXTENDS fbBase
VAR CONSTANT
	TIMEOUT_LOGIC											: TIME 		:= T#20S;
	TIMEOUT_SOCKET											: TIME 		:= T#10S;
	DEL_WRITE_READ											: TIME 		:= T#0MS; //Delay between write and read data
END_VAR
VAR_INPUT
	hSocket													: T_HSOCKET;
	ClrComBuffer											: BOOL := TRUE; //TRUE Clears com buffer before start
	
	pSrc													: POINTER TO BYTE; //Pointer to data source, in case the pointer is empty (0) the FB will only start to wait for data
	cbSrcLen												: UDINT;
	pDest													: POINTER TO BYTE; //Pointer to receive buffer, in case the pointer is empty (0) the FB will only send data and not wait for a response 
	cbDestLen												: UDINT;
END_VAR
VAR_OUTPUT
	RecBytes												: UDINT;
	WinsockErrorId											: E_WinsockError;
END_VAR

VAR
(*  Memory *****************************************************)
	
	ClrBufferLoop											: INT;
	offset													:	UDINT;
(*  Timer ******************************************************)
	Timer1													: Ton;
(*  Trigger ****************************************************)

(*  Blocks *****************************************************)
	SocketSend												: FB_SocketSend := (tTimeout := TIMEOUT_SOCKET);
	SocketReceive											: FB_SocketReceive := (tTimeout := TIMEOUT_SOCKET);
	
(* Cache ******************************************************)
	i														: INT;
END_VAR

(* state machine ********************************************************)
rtExecute(CLK := Execute);

	CASE state OF
	0 : 
		Busy 												:= FALSE;
		IF NOT Execute THEN
			Done 											:= FALSE;
			Error 											:= FALSE;
			ErrorID 										:= 0;
			WinsockErrorId									:= WSOK;
			SocketSend(bExecute	:= FALSE);
			SocketReceive(bExecute := FALSE);
		END_IF
		IF rtExecute.Q THEN
			Busy 											:= TRUE;
			Done											:= FALSE;		
			SocketSend(bExecute	:= FALSE , sSrvNetId	:= '', tTimeout := TIMEOUT_SOCKET);
			SocketReceive(bExecute := FALSE, sSrvNetId	:= '', tTimeout := TIMEOUT_SOCKET);
			IF TRUE			
			THEN
				Error 										:= FALSE;
				ErrorID 									:= 0;
				RecBytes									:= 0;
				offset										:= 0;
				WinsockErrorId								:= WSOK;
				
				Timer1(IN := FALSE);
				ClrBufferLoop								:= 1;

					
				IF pSrc = 0 AND pDest <> 0
				THEN //No command start to received data
					SocketReceive(
						hSocket		:= hSocket, 
						cbLen		:= cbDestLen,  
						pDest		:= pDest, 
						bExecute	:= TRUE);
					state 									:= 4;
				ELSIF pSrc <> 0 AND pDest = 0
				THEN //Just send command, do not wait for response 
					SocketSend(
						hSocket		:= hSocket, 
						cbLen		:= cbSrcLen, 
						pSrc		:= pSrc, 
						bExecute	:= TRUE);
					state									:= 2;
				ELSE //Clear received buffer before starting to send data
					SocketReceive(
						hSocket		:= hSocket, 
						cbLen		:= cbDestLen,  
						pDest		:= pDest, 
						bExecute	:= TRUE);
					state 									:= SEL(ClrComBuffer, 2 , state + 1);
				END_IF
				
			END_IF
		END_IF
		
	1 : // clear communication buffer
		SocketReceive(
			hSocket		:= hSocket, 
			cbLen		:= cbDestLen,  
			pDest		:= pDest, 
			bExecute	:= TRUE);
		IF NOT SocketReceive.bBusy THEN
			IF SocketReceive.nRecBytes > 0
			THEN
				ClrBufferLoop								:= ClrBufferLoop + 1;
			ELSE
				SocketSend(
					hSocket		:= hSocket, 
					cbLen		:= cbSrcLen, 
					pSrc		:= pSrc, 
					bExecute	:= TRUE);
				state										:= state + 1;
			END_IF
			SocketReceive(bExecute := FALSE);
		END_IF

	2 :
		SocketSend(
			hSocket		:= hSocket, 
			cbLen		:= cbSrcLen, 
			pSrc		:= pSrc, 
			bExecute	:= TRUE);
		IF NOT SocketSend.bBusy THEN
			IF NOT SocketSend.bError THEN
				state 										:= SEL(pDest = 0, state + 1 , 0);				
			ELSE
				Error 										:= TRUE;
				ErrorID 									:= SocketSend.nErrId;
				WinsockErrorId								:= ADSERROR_TO_WSERROR(ErrorId);
				
				state 										:= 0;
			END_IF
			SocketSend(bExecute	:= FALSE);
		END_IF

	3 : 
		Timer1(IN := TRUE, PT := DEL_WRITE_READ);
		IF Timer1.Q THEN
			MEMSET(pDest,0,cbDestLen);  //Clear destination
			Timer1(IN := FALSE);
			Timer1(IN := TRUE, PT := TIMEOUT_LOGIC); //Timeout
			state 											:= state + 1;
		END_IF

	4 : 
		Timer1();
		SocketReceive(
			hSocket		:= hSocket, 
			cbLen		:= cbDestLen - offset, 
			pDest		:= pDest + offset, 
			bExecute	:= TRUE);
		IF NOT SocketReceive.bBusy 
		THEN
			IF NOT SocketReceive.bError 
			THEN				
				IF SocketReceive.nRecBytes>0 
				THEN
					RecBytes								:= RecBytes + SocketReceive.nRecBytes;
					offset									:= RecBytes;
					IF RecBytes > cbDestLen 
					THEN //Received data exeeded buffer size
						State								:= 0;
						Error 								:= TRUE;
						ErrorID 							:= E_AdsErr.DEVICE_NOMEMORY;
						WinsockErrorId						:= ADSERROR_TO_WSERROR(ErrorId);	
					ELSE //Just response received data
						state								:= 0;
					END_IF
				ELSIF SocketReceive.nRecBytes = 0 AND RecBytes > 0
				THEN //no more data received 
					state									:= 0;
				ELSIF Timer1.Q 
				THEN
					Timer1(IN := FALSE);
					Error 									:= TRUE;
					ErrorID 								:= E_AdsErr.DEVICE_TIMEOUT;
					WinsockErrorId							:= WSAETIMEDOUT;
					state 									:= 0;
				END_IF	
				
			ELSE
				State										:= 0;
				Error 										:= TRUE;
				ErrorID 									:= SocketReceive.nErrId;
				WinsockErrorId								:= ADSERROR_TO_WSERROR(ErrorId);
			END_IF
	
			SocketReceive(bExecute := FALSE);	// retry as long as state didn't change
		END_IF

	END_CASE

(* reset busy ******************************************************************)
IF Busy AND state = 0 THEN
	Busy 													:= FALSE;
	Done													:= NOT Error;
END_IF
(********************************************************************************)

END_FUNCTION_BLOCK

// POUs/Connectivity/TF6310-TcpServer/DeviceCom/TCPDeviceCom_SendRecString
//FB sends a "command" out and waits for response of the connected device (handshake mode)
//By changing the Fnc the FB mode can be switched into only send or only receive
FUNCTION_BLOCK TCPDeviceCom_SendRecString EXTENDS fbBase
VAR_OUTPUT CONSTANT
	FNC_SEND_REC											:	INT := 0; //Send command and wait for response
	FNC_SEND												:	INT := 1; //Send only
	FNC_REC													:	INT := 2; //Receive only
END_VAR
VAR_INPUT
	Fnc														:	INT(FNC_SEND_REC..FNC_SEND_REC):= FNC_SEND_REC;
	hSocket													: T_HSOCKET;
	ClrComBuffer											: BOOL := TRUE; //TRUE Clears com buffer before start
	Command													: T_MaxString;
	Suffix													: STRING(5) := '$R'; //Will be added to send data and removed from response
END_VAR
VAR_OUTPUT
	ResponseLen												: UDINT;
	Response												: T_MaxString;
	WinsockErrorId											: E_WinsockError;
END_VAR
VAR
	SendRecBytes											:	TCPDeviceCom_SendRecBytes;
	tmpString												:	T_MaxString;
END_VAR
VAR CONSTANT
END_VAR

	IF Execute
		AND NOT SendRecBytes.Execute
	THEN 
		tmpString											:= CONCAT(Command,Suffix);
	END_IF
	
	SendRecBytes(
		Execute:= Execute, 
		hSocket:= hSocket, 
		ClrComBuffer := ClrComBuffer,
		cbSrcLen:= TO_UDINT(LEN(tmpString)), 
		pSrc:= SEL(Command[0] = 0 OR Fnc = FNC_REC , ADR(tmpString),0),
		cbDestLen:= SIZEOF(Response)-1, 
		pDest:= SEL(Fnc = FNC_SEND , ADR(Response),0), 
		Busy=> Busy, 
		Done=> Done, 
		RecBytes=> , 
		Error=> Error, 
		ErrorId=> ErrorId, 
		WinsockErrorId=> WinsockErrorId);
		
	IF SendRecBytes.Done
	THEN
		tmpString											:= ReadStrToSeperator(Suffix,Response);
		IF tmpString[0] <> 0 
		THEN
			Response										:= tmpString;
			ResponseLen										:= TO_UDINT(LEN(Response));
		ELSE
			ResponseLen										:= SendRecBytes.RecBytes;
		END_IF
	END_IF

END_FUNCTION_BLOCK

// POUs/StringHelper/readStrToSeperator
{attribute 'no_check'}
//Returns a string found on the left side of a seperator, empty if seperator is not found
FUNCTION readStrToSeperator : T_MaxString
VAR_INPUT
	Seperator												:	STRING(10) :=';';
	Strline													:	T_MaxString;
END_VAR
VAR_IN_OUT
END_VAR
VAR
	pos														:	INT;
END_VAR

IF strline='' 
THEN
	readStrToSeperator										:= '';
ELSE
	pos 													:= FIND (strline,seperator);
	IF (pos >= 1) 
	THEN
		readStrToSeperator									:= LEFT (strline,pos-1);
	ELSE
		readStrToSeperator									:= '';
	END_IF
END_IF

END_FUNCTION

// POUs/Connectivity/TF6310-TcpServer/TcpBasic/TCPConnectionCtrl
{attribute 'no_check'}
//Helper for TCP Client or Server socket communication communication.
//(Wrapper for Fbs like SocketAccpet,SocketClose,SocketConnect....)
//based on TF6310, required lib: Tc2_TcpIp - see Beckhoff Infosys for more information
FUNCTION_BLOCK TCPConnectionCtrl
VAR_OUTPUT CONSTANT
	FNC_CLIENT_SERVER										:	INT := 0; //Plc runs as client implementation (sending connection request)
	FNC_SERVER_CLIENT										:	INT := 1; //Plc runs as server implementation (acknowledge incomming connetion requests from a client)
END_VAR
VAR_INPUT
	Enable													:	BOOL := FALSE; // FB will be processed as long as enable is TRUE 
	Fnc														: 	INT (FNC_CLIENT_SERVER..FNC_SERVER_CLIENT) := FNC_CLIENT_SERVER;
	SrvNetId												: 	T_AmsNetId := ''; //AmsNet id for TcpIp Server instance - '' for local 
	SrvLocalHost											:	T_IPv4Addr := '127.0.0.1';		 //IP-Adress of local ip-adapter used for server communication
	SrvLocalPort											:	UDINT;			//IP-Port of local ip-adapter used for server communication
	SrvAcceptMode											: 	E_SocketAcceptMode :=	eACCEPT_ALL; (* 	eACCEPT_ALL, Accept connection to all remote clients
																							eACCEPT_SEL_HOST,  Accept connection TO selected host address
																							eACCEPT_SEL_PORT,  Accept connection to selected port address 
																							eACCEPT_SEL_HOeSTATE.PORT  Accept connection to selected host and port address *)
	RemoteHost 												: 	T_IPv4Addr := '' ;//Remote/Client Ip-Adress used for Client/Server communication - Empty for an unspecified adapter
	RemotePort												: 	UDINT := 0; //Remote/Client socket port used for Client/Server communication - Empty for an unspecified port
	PT_Reconnect											:	TIME := T#30S; //In Server mode tReconnet can be set to 1ms, as a client the tReconnect value should not be set too low, since timeout periods of > 30 s may occur in the event of a network interruption. If the value is too low, command execution would be interrupted prematurely, and ADS error code 1861 (timeout elapsed) would be returned instead of the Winsocket error WSAETIMEDOUT.
	PT_LinkStatus											:	TIME := T#5S; //Cycle time to check adapter link status T#0ms = off	

	EnableDebugMode											:	BOOL := FALSE; //Write debug information into twincat logger
	CloseAllSocket											:	BOOL := TRUE; //Close all socket if server will be diabled - FALSE = close only connected port
END_VAR                 									
VAR_OUTPUT              									
	hSocket													: 	T_HSOCKET ; //
	hSocketText												:	STRING(80); //
	Connected												:	BOOL; (* Connection is current running *)
	LinkNOK													:	BOOL; //TRUE = Link not ok			
	Reconnecting											:	BOOL; //Reconnet because of new incomming connection		
	ConnState												:	E_SocketConnectionState; // Socket connection state enum - see TF6310 documentation for further information
	Busy													:	BOOL;	// Busy is TRUE at the rising edge of Enable and stays TRUE as long as the FB is performing any action. 
	Error													:	BOOL;	// Rising edge of Error informs that an error occurred during the execution of the Function Block 
{attribute 'displaymode':='hex'}
	ErrorId													:	UDINT;	// Error identification - see ADS return codes and TF6310 documentation at Beckhoff infosys for further information 
	WinsockErrorId											:	E_WinsockError; // Winsocket error enum - see TF6310 documentation for further information
END_VAR
VAR
END_VAR
VAR
(* local variables ************************************************************)
	ReadyToEnable											:	BOOL;
	hServer													:	T_HSERVER;

(* Trigger **********************************************************)

(* Timer ******************************************************************)
	LinkDetectionTimer										:	TON;
	
(* Insatcnced ***************************************************************)	
	IpAdapterLinkStatus										:	FB_IpAdapterGetLinkStatus := (sSrvNetId := '', ttimeout := DEFAULT_ADS_TIMEOUT) ;		
	Server													:	 FB_ServerClientConnection;
	Server2													:	 FB_ServerClientConnection;
	Client													:	 FB_ClientServerConnection;

(* Dummys **********************************************************)

END_VAR

(* Link status ***********************************************************)	
	LinkDetectionTimer( 
		IN := Enable
			AND PT_LinkStatus > T#0MS
			AND NOT LinkDetectionTimer.Q 	
			AND NOT IpAdapterLinkStatus.bBusy,
		PT := PT_LinkStatus);
	
	IpAdapterLinkStatus(
		sSrvNetId		:= , 
		sLocalHost		:= hSocket.localAddr.sAddr, 
		bExecute		:= LinkDetectionTimer.Q OR IpAdapterLinkStatus.bBusy ,
		tTimeout		:=, 
		bBusy			=> , 
		bError			=> , 
		nErrId			=> , 
		bLinkError		=> );
	
	IF NOT IpAdapterLinkStatus.bBusy
		AND IpAdapterLinkStatus.bExecute
	THEN
		LinkNOK												:= 	IpAdapterLinkStatus.bLinkError;
	END_IF


(* Ready to enable ******************************************************)
	//Enable and disabled server to closed old connection if new incoming connection occured
	ReadyToEnable											:= Enable 
																AND NOT IpAdapterLinkStatus.bLinkError
																AND NOT Error;
																
(* Execute ********************************************************************************)	
IF Fnc = FNC_SERVER_CLIENT AND NOT Client.bBusy
	OR Server.bBusy OR Server2.bbusy
THEN //accept client request
(* run server ************************************************************)																																											
	_RunAsServer();
ELSE
	_RunAsClient();
END_IF

(**************************************************************************************)

METHOD PRIVATE _RunAsClient : BOOL
VAR_INPUT
END_VAR
	Client(
		sSrvNetID		:= SrvNetId,
		nMode			:= SEL(EnableDebugMode,0,CONNECT_MODE_ENABLEDBG),
		sRemoteHost		:= RemoteHost,
		nRemotePort		:= RemotePort,
		bEnable			:= ReadyToEnable AND Fnc = FNC_CLIENT_SERVER,
		tReconnect		:= PT_Reconnect,
		bBusy			=> Busy,
		bError			=> ,
		nErrId			=> ,
		hSocket			=> hSocket,
		eSTATE			=> ConnState);

	Connected 												:= hSocket.handle <> 0 AND ConnState = E_SocketConnectionState.eSOCKET_CONNECTED;
	hSocketText												:= HSOCKET_TO_STRING(hSocket);
	
	IF Error
	THEN
		IF NOT Enable
		THEN
			Error											:= FALSE;
			ErrorId											:= 0;
			WinsockErrorId									:= WSOK;		
		END_IF
	ELSIF Client.bError
	THEN
		Error												:= TRUE;
		IF Client.nErrId >= 16#80070000
		THEN
			ErrorId											:= E_AdsErr.CLIENT_W32ERROR;
			WinsockErrorId									:= ADSERROR_TO_WSERROR(Client.nErrId);
		ELSE                    								
			ErrorId											:= Client.nErrId;
			WinsockErrorId									:= WSOK;
		END_IF
	END_IF
	
	_RunAsClient											:= Connected;
END_METHOD

METHOD _RunAsServer : BOOL
VAR_INPUT
END_VAR
(* Init Serverhandle *********************************)
	IF NOT Connected AND ReadyToEnable
		OR ConnState <> E_SocketConnectionState.eSOCKET_DISCONNECTED AND NOT Enable
		OR Reconnecting
	THEN
		F_CreateServerHnd(
			sSrvNetID		:= SrvNetId,
			sLocalHost		:= SrvLocalHost,
			nLocalPort		:= SrvLocalPort,
			nMode			:= SEL(EnableDebugMode,0,CONNECT_MODE_ENABLEDBG) OR SEL(CloseAllSocket OR Reconnecting,0,LISTEN_MODE_CLOSEALL),
			bEnable			:= Server.bEnable OR Server2.bEnable,
			hServer			:= hServer);
	END_IF

(* Call Server **************************************)
	Server(
		eMode			:= SrvAcceptMode,
		sRemoteHost		:= RemoteHost,
		nRemotePort		:= RemotePort,
		bEnable			:= ,
		tReconnect		:= PT_Reconnect,
		hServer			:= hServer,
		bBusy			=> ,
		bError			=> ,
		nErrID			=> ,
		hSocket			=> ,
		eSTATE			=> );
		
		
	Server2(
		eMode			:= SrvAcceptMode,
		sRemoteHost		:= RemoteHost,
		nRemotePort		:= RemotePort,
		bEnable			:= ,
		tReconnect		:= PT_Reconnect,
		hServer			:= hServer,
		bBusy			=> ,
		bError			=> ,
		nErrID			=> ,
		hSocket			=> ,
		eSTATE			=> );
	
	//Control server enable 	
	IF NOT ReadyToEnable
	THEN
		Server2.bEnable										:= FALSE;
		Server.bEnable										:= FALSE;
		ConnState											:= eSOCKET_DISCONNECTED;
		hSocket.handle										:= 0;		
		
	ELSIF Server.hSocket.handle <> 0 AND Server2.hSocket.handle	<> 0
	THEN
		Server.bEnable										:= Server.hSocket.handle <> hSocket.handle;
		Server2.bEnable										:= Server2.hSocket.handle <> hSocket.handle;
		ConnState											:= eSOCKET_DISCONNECTED;	
	ELSif Server.hSocket.handle <> 0
	THEN
		hSocket												:= Server.hSocket;	
		ConnState											:= Server.eState;
		Server2.bEnable										:= Server2.hSocket.handle = 0;	
	ELSIF Server2.hSocket.handle <> 0
	THEN
		hSocket												:= Server2.hSocket;	
		ConnState											:= Server2.eState;
		Server.bEnable										:= Server.hSocket.handle = 0;	
	ELSE
		ConnState											:= eSOCKET_DISCONNECTED;
		hSocket.handle										:= 0;		
		Server.bEnable										:= Server.hSocket.handle = 0;
		Server2.bEnable										:= Server2.hSocket.handle = 0;					
	END_IF			
	
(* Error check *******************************************************)
	IF Error
	THEN
		IF NOT Enable
		THEN
			Error											:= FALSE;
			ErrorId											:= 0;
			WinsockErrorId									:= WSOK;		
		END_IF
		
	ELSIF LinkNOK AND Connected
	THEN
		Error												:= TRUE;
		ErrorID												:= 16#80070000 OR 16#00002742;
		WinsockErrorId										:= ADSERROR_TO_WSERROR(ErrorID);
		
